SPLINE
SPL {X  -126.418, Y  +769.557, Z    +0.000, E1  +417.118, E3 -55794.219}
SPL {X  -145.244, Y  +738.589, Z    +0.000, E1  +410.405, E3 -55807.461}
SPL {X  -150.151, Y  +726.741, Z    +0.000, E1  +406.068, E3 -55810.388}
SPL {X  -156.642, Y  +704.059, Z    +0.000, E1  +393.659, E3 -55814.017}
SPL {X  -159.317, Y  +686.157, Z    +0.000, E1  +378.660, E3 -55815.507}
SPL {X  -159.973, Y  +673.799, Z    +0.000, E1  +365.345, E3 -55815.956}
SPL {X  -159.990, Y  +669.500, Z    +0.000, E1  +360.000, E3 -55815.996}
SPL {X  -159.990, Y  +667.794, Z    +0.000, E1  +355.745, E3 -55816.007}
SPL {X  -159.990, Y  +664.091, Z    +0.000, E1  +345.072, E3 -55816.079}
SPL {X  -159.990, Y  +659.599, Z    +0.000, E1  +331.984, E3 -55816.250}
SPL {X  -159.990, Y  +652.711, Z    +0.000, E1  +315.707, E3 -55816.729}
SPL {X  -159.990, Y  +640.730, Z    +0.000, E1  +299.703, E3 -55818.078}
SPL {X  -159.990, Y  +620.478, Z    +0.000, E1  +289.974, E3 -55821.891}
SPL {X  -159.990, Y  +573.021, Z    +0.000, E1  +285.381, E3 -55835.835}
SPL {X  -155.476, Y  +344.766, Z    +0.000, E1  +283.975, E3 -55927.806}
SPL {X  -153.405, Y  +337.073, Z    +0.000, E1  +284.153, E3 -55933.861}
SPL {X  -150.223, Y  +327.456, Z    +0.000, E1  +284.427, E3 -55941.947}
SPL {X  -136.549, Y  +299.126, Z    +0.000, E1  +282.463, E3 -55934.837}
ENDSPLINE

SPLINE
SPL {X  -136.626, Y  +299.252, Z    +0.000, E1  +283.686, E3 -55946.487}
ENDSPLINE

SPLINE
SPL {X  -135.890, Y  +298.057, Z    +0.000, E1  +284.960, E3 -55957.836}
SPL {X  -134.349, Y  +295.626, Z    +0.000, E1  +285.678, E3 -55964.683}
SPL {X  -131.287, Y  +291.064, Z    +0.000, E1  +286.028, E3 -55969.496}
SPL {X  -128.265, Y  +286.871, Z    +0.000, E1  +286.387, E3 -55973.952}
SPL {X  -125.161, Y  +282.843, Z    +0.000, E1  +286.768, E3 -55978.224}
SPL {X  -122.038, Y  +279.042, Z    +0.000, E1  +287.168, E3 -55982.204}
SPL {X  -118.642, Y  +275.165, Z    +0.000, E1  +287.619, E3 -55986.167}
SPL {X   -66.040, Y  +236.776, Z    +0.000, E1  +304.306, E3 -56147.530}
ENDSPLINE

SPLINE
SPL {X  -127.452, Y  +285.790, Z    +0.000, E1  +303.409, E3 -56321.476}
SPL {X  -148.001, Y  +321.733, Z    +0.000, E1  +312.190, E3 -56335.579}
SPL {X  -154.604, Y  +341.337, Z    +0.000, E1  +321.370, E3 -56339.353}
SPL {X  -158.135, Y  +358.205, Z    +0.000, E1  +333.016, E3 -56341.302}
SPL {X  -159.602, Y  +371.361, Z    +0.000, E1  +345.165, E3 -56342.198}
SPL {X  -159.981, Y  +380.818, Z    +0.000, E1  +355.488, E3 -56342.476}
SPL {X  -159.990, Y  +384.681, Z    +0.000, E1  +360.222, E3 -56342.505}
SPL {X  -159.990, Y  +389.079, Z    +0.000, E1  +372.017, E3 -56342.568}
SPL {X  -159.990, Y  +394.216, Z    +0.000, E1  +387.062, E3 -56342.760}
SPL {X  -159.990, Y  +401.720, Z    +0.000, E1  +404.434, E3 -56343.303}
SPL {X  -159.990, Y  +414.231, Z    +0.000, E1  +420.575, E3 -56344.832}
SPL {X  -159.990, Y  +462.953, Z    +0.000, E1  +433.611, E3 -56356.571}
SPL {X  -153.839, Y  +715.436, Z    +0.000, E1  +435.884, E3 -56459.002}
SPL {X  -149.923, Y  +727.355, Z    +0.000, E1  +435.515, E3 -56469.112}
SPL {X  -145.995, Y  +736.939, Z    +0.000, E1  +435.150, E3 -56477.846}
SPL {X  -142.305, Y  +744.618, Z    +0.000, E1  +434.773, E3 -56485.290}
SPL {X  -139.557, Y  +749.735, Z    +0.000, E1  +434.483, E3 -56490.439}
SPL {X  -136.371, Y  +755.165, Z    +0.000, E1  +434.152, E3 -56495.984}
SPL {X  -133.102, Y  +760.274, Z    +0.000, E1  +433.777, E3 -56501.369}
SPL {X  -128.975, Y  +766.169, Z    +0.000, E1  +433.313, E3 -56507.645}
SPL {X  -124.947, Y  +771.425, Z    +0.000, E1  +432.782, E3 -56513.338}
SPL {X  -121.698, Y  +775.357, Z    +0.000, E1  +432.353, E3 -56517.532}
SPL {X  -118.622, Y  +778.858, Z    +0.000, E1  +431.924, E3 -56521.158}
SPL {X   -66.171, Y  +817.165, Z    +0.000, E1  +416.016, E3 -56672.517}
ENDSPLINE

SPLINE
SPL {X  -126.418, Y  +769.557, Z    +0.000, E1  +417.118, E3 -56855.758}
SPL {X  -145.244, Y  +738.589, Z    +0.000, E1  +410.405, E3 -56868.999}
SPL {X  -150.151, Y  +726.741, Z    +0.000, E1  +406.068, E3 -56871.926}
SPL {X  -156.642, Y  +704.059, Z    +0.000, E1  +393.659, E3 -56875.555}
SPL {X  -159.317, Y  +686.157, Z    +0.000, E1  +378.660, E3 -56877.046}
SPL {X  -159.973, Y  +673.799, Z    +0.000, E1  +365.345, E3 -56877.494}
SPL {X  -159.990, Y  +669.500, Z    +0.000, E1  +360.000, E3 -56877.534}
SPL {X  -159.990, Y  +667.794, Z    +0.000, E1  +355.745, E3 -56877.546}
SPL {X  -159.990, Y  +664.091, Z    +0.000, E1  +345.072, E3 -56877.618}
SPL {X  -159.990, Y  +658.301, Z    +0.000, E1  +328.717, E3 -56877.870}
SPL {X  -159.990, Y  +650.845, Z    +0.000, E1  +312.108, E3 -56878.415}
SPL {X  -159.990, Y  +640.730, Z    +0.000, E1  +299.703, E3 -56879.617}
SPL {X  -159.990, Y  +620.478, Z    +0.000, E1  +289.974, E3 -56883.430}
SPL {X  -159.990, Y  +573.021, Z    +0.000, E1  +285.381, E3 -56897.374}
SPL {X  -154.165, Y  +339.724, Z    +0.000, E1  +284.073, E3 -56993.221}
SPL {X  -150.223, Y  +327.456, Z    +0.000, E1  +284.427, E3 -57003.486}
SPL {X  -136.549, Y  +299.126, Z    +0.000, E1  +282.463, E3 -56996.376}
ENDSPLINE

SPLINE
SPL {X  -136.862, Y  +299.641, Z    +0.000, E1  +283.396, E3 -57005.018}
ENDSPLINE

SPLINE
SPL {X  -136.434, Y  +298.938, Z    +0.000, E1  +284.018, E3 -57010.909}
SPL {X  -135.890, Y  +298.057, Z    +0.000, E1  +284.960, E3 -57019.375}
SPL {X  -134.349, Y  +295.626, Z    +0.000, E1  +285.678, E3 -57026.222}
SPL {X  -131.287, Y  +291.064, Z    +0.000, E1  +286.028, E3 -57031.034}
SPL {X  -128.265, Y  +286.871, Z    +0.000, E1  +286.387, E3 -57035.490}
SPL {X  -125.161, Y  +282.843, Z    +0.000, E1  +286.768, E3 -57039.762}
SPL {X  -122.038, Y  +279.042, Z    +0.000, E1  +287.168, E3 -57043.742}
SPL {X  -118.642, Y  +275.165, Z    +0.000, E1  +287.619, E3 -57047.705}
SPL {X   -66.040, Y  +236.776, Z    +0.000, E1  +304.306, E3 -57209.069}
ENDSPLINE

SPLINE
SPL {X  -127.452, Y  +285.790, Z    +0.000, E1  +303.409, E3 -57383.014}
SPL {X  -148.001, Y  +321.733, Z    +0.000, E1  +312.190, E3 -57397.118}
SPL {X  -154.604, Y  +341.337, Z    +0.000, E1  +321.370, E3 -57400.891}
SPL {X  -158.135, Y  +358.205, Z    +0.000, E1  +333.016, E3 -57402.841}
SPL {X  -159.602, Y  +371.361, Z    +0.000, E1  +345.165, E3 -57403.737}
SPL {X  -159.981, Y  +380.818, Z    +0.000, E1  +355.488, E3 -57404.015}
SPL {X  -159.990, Y  +384.681, Z    +0.000, E1  +360.222, E3 -57404.044}
SPL {X  -159.990, Y  +389.079, Z    +0.000, E1  +372.017, E3 -57404.107}
SPL {X  -159.990, Y  +394.216, Z    +0.000, E1  +387.062, E3 -57404.299}
SPL {X  -159.990, Y  +399.855, Z    +0.000, E1  +400.916, E3 -57404.670}
SPL {X  -159.990, Y  +405.475, Z    +0.000, E1  +411.039, E3 -57405.187}
SPL {X  -159.990, Y  +414.231, Z    +0.000, E1  +420.575, E3 -57406.371}
SPL {X  -159.990, Y  +462.953, Z    +0.000, E1  +433.611, E3 -57418.110}
SPL {X  -153.839, Y  +715.436, Z    +0.000, E1  +435.884, E3 -57520.540}
SPL {X  -148.840, Y  +730.182, Z    +0.000, E1  +435.434, E3 -57533.117}
SPL {X  -143.409, Y  +742.426, Z    +0.000, E1  +434.905, E3 -57544.629}
SPL {X  -139.557, Y  +749.735, Z    +0.000, E1  +434.483, E3 -57551.977}
SPL {X  -136.371, Y  +755.165, Z    +0.000, E1  +434.152, E3 -57557.523}
SPL {X  -133.102, Y  +760.274, Z    +0.000, E1  +433.777, E3 -57562.908}
SPL {X  -128.975, Y  +766.169, Z    +0.000, E1  +433.313, E3 -57569.183}
SPL {X  -124.947, Y  +771.425, Z    +0.000, E1  +432.782, E3 -57574.876}
SPL {X  -121.698, Y  +775.357, Z    +0.000, E1  +432.353, E3 -57579.071}
SPL {X  -118.622, Y  +778.858, Z    +0.000, E1  +431.924, E3 -57582.697}
SPL {X   -66.171, Y  +817.165, Z    +0.000, E1  +416.016, E3 -57734.055}
ENDSPLINE

SPLINE
SPL {X  -126.418, Y  +769.557, Z    +0.000, E1  +417.118, E3 -57917.296}
SPL {X  -145.244, Y  +738.589, Z    +0.000, E1  +410.405, E3 -57930.538}
SPL {X  -150.151, Y  +726.741, Z    +0.000, E1  +406.068, E3 -57933.464}
SPL {X  -156.642, Y  +704.059, Z    +0.000, E1  +393.659, E3 -57937.094}
SPL {X  -159.317, Y  +686.157, Z    +0.000, E1  +378.660, E3 -57938.584}
SPL {X  -159.973, Y  +673.799, Z    +0.000, E1  +365.345, E3 -57939.033}
SPL {X  -159.990, Y  +669.500, Z    +0.000, E1  +360.000, E3 -57939.073}
SPL {X  -159.990, Y  +667.794, Z    +0.000, E1  +355.745, E3 -57939.084}
SPL {X  -159.990, Y  +664.091, Z    +0.000, E1  +345.072, E3 -57939.156}
SPL {X  -159.990, Y  +658.301, Z    +0.000, E1  +328.717, E3 -57939.409}
SPL {X  -159.990, Y  +650.845, Z    +0.000, E1  +312.108, E3 -57939.954}
SPL {X  -159.990, Y  +640.730, Z    +0.000, E1  +299.703, E3 -57941.155}
SPL {X  -159.990, Y  +620.478, Z    +0.000, E1  +289.974, E3 -57944.968}
SPL {X  -159.990, Y  +573.021, Z    +0.000, E1  +285.381, E3 -57958.912}
SPL {X  -154.165, Y  +339.724, Z    +0.000, E1  +284.073, E3 -58054.759}
SPL {X  -150.223, Y  +327.456, Z    +0.000, E1  +284.427, E3 -58065.024}
SPL {X  -136.549, Y  +299.126, Z    +0.000, E1  +282.463, E3 -58057.914}
ENDSPLINE

SPLINE
SPL {X  -136.862, Y  +299.641, Z    +0.000, E1  +283.396, E3 -58066.556}
ENDSPLINE

SPLINE
SPL {X  -136.434, Y  +298.938, Z    +0.000, E1  +284.018, E3 -58072.447}
SPL {X  -135.890, Y  +298.057, Z    +0.000, E1  +284.960, E3 -58080.913}
SPL {X  -134.349, Y  +295.626, Z    +0.000, E1  +285.678, E3 -58087.760}
SPL {X  -131.287, Y  +291.064, Z    +0.000, E1  +286.028, E3 -58092.573}
SPL {X  -128.265, Y  +286.871, Z    +0.000, E1  +286.387, E3 -58097.029}
SPL {X  -125.161, Y  +282.843, Z    +0.000, E1  +286.768, E3 -58101.301}
SPL {X  -122.038, Y  +279.042, Z    +0.000, E1  +287.168, E3 -58105.281}
SPL {X  -118.642, Y  +275.165, Z    +0.000, E1  +287.619, E3 -58109.244}
SPL {X   -66.040, Y  +236.776, Z    +0.000, E1  +304.306, E3 -58270.607}
ENDSPLINE

SPLINE
SPL {X  -127.452, Y  +285.790, Z    +0.000, E1  +303.409, E3 -58444.552}
SPL {X  -148.001, Y  +321.733, Z    +0.000, E1  +312.190, E3 -58458.656}
SPL {X  -154.604, Y  +341.337, Z    +0.000, E1  +321.370, E3 -58462.430}
SPL {X  -158.135, Y  +358.205, Z    +0.000, E1  +333.016, E3 -58464.379}
SPL {X  -159.602, Y  +371.361, Z    +0.000, E1  +345.165, E3 -58465.275}
SPL {X  -159.981, Y  +380.818, Z    +0.000, E1  +355.488, E3 -58465.553}
SPL {X  -159.990, Y  +384.681, Z    +0.000, E1  +360.222, E3 -58465.582}
SPL {X  -159.990, Y  +389.079, Z    +0.000, E1  +372.017, E3 -58465.645}
SPL {X  -159.990, Y  +394.216, Z    +0.000, E1  +387.062, E3 -58465.837}
SPL {X  -159.990, Y  +399.855, Z    +0.000, E1  +400.916, E3 -58466.208}
SPL {X  -159.990, Y  +405.475, Z    +0.000, E1  +411.039, E3 -58466.725}
SPL {X  -159.990, Y  +414.231, Z    +0.000, E1  +420.575, E3 -58467.909}
SPL {X  -159.990, Y  +462.953, Z    +0.000, E1  +433.611, E3 -58479.648}
SPL {X  -153.839, Y  +715.436, Z    +0.000, E1  +435.884, E3 -58582.079}
SPL {X  -148.840, Y  +730.182, Z    +0.000, E1  +435.434, E3 -58594.655}
SPL {X  -143.409, Y  +742.426, Z    +0.000, E1  +434.905, E3 -58606.167}
SPL {X  -139.557, Y  +749.735, Z    +0.000, E1  +434.483, E3 -58613.515}
SPL {X  -136.371, Y  +755.165, Z    +0.000, E1  +434.152, E3 -58619.061}
SPL {X  -133.102, Y  +760.274, Z    +0.000, E1  +433.777, E3 -58624.446}
SPL {X  -128.975, Y  +766.169, Z    +0.000, E1  +433.313, E3 -58630.722}
SPL {X  -124.947, Y  +771.425, Z    +0.000, E1  +432.782, E3 -58636.415}
SPL {X  -121.698, Y  +775.357, Z    +0.000, E1  +432.353, E3 -58640.609}
SPL {X  -118.622, Y  +778.858, Z    +0.000, E1  +431.924, E3 -58644.235}
SPL {X   -66.171, Y  +817.165, Z    +0.000, E1  +416.016, E3 -58795.593}
ENDSPLINE

SPLINE
SPL {X  -126.418, Y  +769.557, Z    +0.000, E1  +417.118, E3 -58978.835}
SPL {X  -145.244, Y  +738.589, Z    +0.000, E1  +410.405, E3 -58992.076}
SPL {X  -150.151, Y  +726.741, Z    +0.000, E1  +406.068, E3 -58995.003}
SPL {X  -156.642, Y  +704.059, Z    +0.000, E1  +393.659, E3 -58998.632}
SPL {X  -159.317, Y  +686.157, Z    +0.000, E1  +378.660, E3 -59000.123}
SPL {X  -159.973, Y  +673.799, Z    +0.000, E1  +365.345, E3 -59000.571}
SPL {X  -159.990, Y  +669.500, Z    +0.000, E1  +360.000, E3 -59000.611}
SPL {X  -159.990, Y  +667.794, Z    +0.000, E1  +355.745, E3 -59000.623}
SPL {X  -159.990, Y  +664.091, Z    +0.000, E1  +345.072, E3 -59000.695}
SPL {X  -159.990, Y  +658.301, Z    +0.000, E1  +328.717, E3 -59000.947}
SPL {X  -159.990, Y  +650.845, Z    +0.000, E1  +312.108, E3 -59001.492}
SPL {X  -159.990, Y  +640.730, Z    +0.000, E1  +299.703, E3 -59002.693}
SPL {X  -159.990, Y  +620.478, Z    +0.000, E1  +289.974, E3 -59006.507}
SPL {X  -159.990, Y  +573.021, Z    +0.000, E1  +285.381, E3 -59020.451}
SPL {X  -154.165, Y  +339.724, Z    +0.000, E1  +284.073, E3 -59116.298}
SPL {X  -150.223, Y  +327.456, Z    +0.000, E1  +284.427, E3 -59126.562}
SPL {X  -136.549, Y  +299.126, Z    +0.000, E1  +282.463, E3 -59119.452}
ENDSPLINE

SPLINE
SPL {X  -136.862, Y  +299.641, Z    +0.000, E1  +283.396, E3 -59128.094}
ENDSPLINE

SPLINE
SPL {X  -136.434, Y  +298.938, Z    +0.000, E1  +284.018, E3 -59133.986}
SPL {X  -135.890, Y  +298.057, Z    +0.000, E1  +284.960, E3 -59142.452}
SPL {X  -134.349, Y  +295.626, Z    +0.000, E1  +285.678, E3 -59149.299}
SPL {X  -131.287, Y  +291.064, Z    +0.000, E1  +286.028, E3 -59154.111}
SPL {X  -128.265, Y  +286.871, Z    +0.000, E1  +286.387, E3 -59158.567}
SPL {X  -125.161, Y  +282.843, Z    +0.000, E1  +286.768, E3 -59162.839}
SPL {X  -122.038, Y  +279.042, Z    +0.000, E1  +287.168, E3 -59166.819}
SPL {X  -118.642, Y  +275.165, Z    +0.000, E1  +287.619, E3 -59170.782}
SPL {X   -66.040, Y  +236.776, Z    +0.000, E1  +304.306, E3 -59332.146}
ENDSPLINE

SPLINE
SPL {X  -127.452, Y  +285.790, Z    +0.000, E1  +303.409, E3 -59506.091}
SPL {X  -151.591, Y  +331.344, Z    +0.000, E1  +316.130, E3 -59522.190}
SPL {X  -158.135, Y  +358.205, Z    +0.000, E1  +333.016, E3 -59525.918}
SPL {X  -159.602, Y  +371.361, Z    +0.000, E1  +345.165, E3 -59526.814}
SPL {X  -159.981, Y  +380.818, Z    +0.000, E1  +355.488, E3 -59527.092}
SPL {X  -159.990, Y  +384.681, Z    +0.000, E1  +360.222, E3 -59527.121}
SPL {X  -159.990, Y  +387.626, Z    +0.000, E1  +368.190, E3 -59527.149}
SPL {X  -159.990, Y  +390.340, Z    +0.000, E1  +375.987, E3 -59527.214}
SPL {X  -159.990, Y  +394.216, Z    +0.000, E1  +387.062, E3 -59527.375}
SPL {X  -159.990, Y  +399.855, Z    +0.000, E1  +400.916, E3 -59527.747}
SPL {X  -159.990, Y  +405.475, Z    +0.000, E1  +411.039, E3 -59528.263}
SPL {X  -159.990, Y  +414.231, Z    +0.000, E1  +420.575, E3 -59529.448}
SPL {X  -159.990, Y  +462.953, Z    +0.000, E1  +433.611, E3 -59541.187}
SPL {X  -153.839, Y  +715.436, Z    +0.000, E1  +435.884, E3 -59643.617}
SPL {X  -148.840, Y  +730.182, Z    +0.000, E1  +435.434, E3 -59656.194}
SPL {X  -143.409, Y  +742.426, Z    +0.000, E1  +434.905, E3 -59667.706}
SPL {X  -139.557, Y  +749.735, Z    +0.000, E1  +434.483, E3 -59675.054}
SPL {X  -136.371, Y  +755.165, Z    +0.000, E1  +434.152, E3 -59680.600}
SPL {X  -133.102, Y  +760.274, Z    +0.000, E1  +433.777, E3 -59685.985}
SPL {X  -128.975, Y  +766.169, Z    +0.000, E1  +433.313, E3 -59692.260}
SPL {X  -124.947, Y  +771.425, Z    +0.000, E1  +432.782, E3 -59697.953}
SPL {X  -121.698, Y  +775.357, Z    +0.000, E1  +432.353, E3 -59702.148}
SPL {X  -118.622, Y  +778.858, Z    +0.000, E1  +431.924, E3 -59705.774}
SPL {X   -66.171, Y  +817.165, Z    +0.000, E1  +416.016, E3 -59857.132}
ENDSPLINE

SPLINE
SPL {X  -126.418, Y  +769.557, Z    +0.000, E1  +417.118, E3 -60040.373}
SPL {X  -148.476, Y  +731.097, Z    +0.000, E1  +407.824, E3 -60055.529}
SPL {X  -156.642, Y  +704.059, Z    +0.000, E1  +393.659, E3 -60060.171}
SPL {X  -159.317, Y  +686.157, Z    +0.000, E1  +378.660, E3 -60061.661}
SPL {X  -159.907, Y  +676.666, Z    +0.000, E1  +368.555, E3 -60062.059}
SPL {X  -159.990, Y  +669.586, Z    +0.000, E1  +360.216, E3 -60062.149}
SPL {X  -159.990, Y  +667.794, Z    +0.000, E1  +355.745, E3 -60062.161}
SPL {X  -159.990, Y  +664.091, Z    +0.000, E1  +345.072, E3 -60062.233}
SPL {X  -159.990, Y  +659.599, Z    +0.000, E1  +331.984, E3 -60062.404}
SPL {X  -159.990, Y  +652.711, Z    +0.000, E1  +315.707, E3 -60062.883}
SPL {X  -159.990, Y  +640.730, Z    +0.000, E1  +299.703, E3 -60064.232}
SPL {X  -159.990, Y  +620.478, Z    +0.000, E1  +289.974, E3 -60068.045}
SPL {X  -159.990, Y  +573.021, Z    +0.000, E1  +285.381, E3 -60081.989}
SPL {X  -154.165, Y  +339.724, Z    +0.000, E1  +284.073, E3 -60177.836}
SPL {X  -150.571, Y  +328.416, Z    +0.000, E1  +284.401, E3 -60187.281}
SPL {X  -148.206, Y  +322.236, Z    +0.000, E1  +284.635, E3 -60192.826}
SPL {X  -136.549, Y  +299.126, Z    +0.000, E1  +282.463, E3 -60180.991}
ENDSPLINE

SPLINE
SPL {X  -136.862, Y  +299.641, Z    +0.000, E1  +283.396, E3 -60189.633}
ENDSPLINE

SPLINE
SPL {X  -136.434, Y  +298.938, Z    +0.000, E1  +284.018, E3 -60195.524}
SPL {X  -135.890, Y  +298.057, Z    +0.000, E1  +284.960, E3 -60203.990}
SPL {X  -134.349, Y  +295.626, Z    +0.000, E1  +285.678, E3 -60210.837}
SPL {X  -131.287, Y  +291.064, Z    +0.000, E1  +286.028, E3 -60215.650}
SPL {X  -128.265, Y  +286.871, Z    +0.000, E1  +286.387, E3 -60220.106}
SPL {X  -125.161, Y  +282.843, Z    +0.000, E1  +286.768, E3 -60224.378}
SPL {X  -122.038, Y  +279.042, Z    +0.000, E1  +287.168, E3 -60228.357}
SPL {X  -118.642, Y  +275.165, Z    +0.000, E1  +287.619, E3 -60232.321}
SPL {X   -66.040, Y  +236.776, Z    +0.000, E1  +304.306, E3 -60393.684}
ENDSPLINE

SPLINE
SPL {X  -127.452, Y  +285.790, Z    +0.000, E1  +303.409, E3 -60567.629}
SPL {X  -151.591, Y  +331.344, Z    +0.000, E1  +316.130, E3 -60583.729}
SPL {X  -158.135, Y  +358.205, Z    +0.000, E1  +333.016, E3 -60587.456}
SPL {X  -159.602, Y  +371.361, Z    +0.000, E1  +345.165, E3 -60588.352}
SPL {X  -159.981, Y  +380.818, Z    +0.000, E1  +355.488, E3 -60588.630}
SPL {X  -159.990, Y  +384.681, Z    +0.000, E1  +360.222, E3 -60588.659}
SPL {X  -159.990, Y  +389.079, Z    +0.000, E1  +372.017, E3 -60588.722}
SPL {X  -159.990, Y  +394.216, Z    +0.000, E1  +387.062, E3 -60588.914}
SPL {X  -159.990, Y  +399.855, Z    +0.000, E1  +400.916, E3 -60589.285}
SPL {X  -159.990, Y  +405.475, Z    +0.000, E1  +411.039, E3 -60589.802}
SPL {X  -159.990, Y  +414.231, Z    +0.000, E1  +420.575, E3 -60590.986}
SPL {X  -159.990, Y  +462.953, Z    +0.000, E1  +433.611, E3 -60602.725}
SPL {X  -153.839, Y  +715.436, Z    +0.000, E1  +435.884, E3 -60705.156}
SPL {X  -148.840, Y  +730.182, Z    +0.000, E1  +435.434, E3 -60717.732}
SPL {X  -143.409, Y  +742.426, Z    +0.000, E1  +434.905, E3 -60729.244}
SPL {X  -139.557, Y  +749.735, Z    +0.000, E1  +434.483, E3 -60736.592}
SPL {X  -136.371, Y  +755.165, Z    +0.000, E1  +434.152, E3 -60742.138}
SPL {X  -133.102, Y  +760.274, Z    +0.000, E1  +433.777, E3 -60747.523}
SPL {X  -128.975, Y  +766.169, Z    +0.000, E1  +433.313, E3 -60753.799}
SPL {X  -124.947, Y  +771.425, Z    +0.000, E1  +432.782, E3 -60759.492}
SPL {X  -121.698, Y  +775.357, Z    +0.000, E1  +432.353, E3 -60763.686}
SPL {X  -118.622, Y  +778.858, Z    +0.000, E1  +431.924, E3 -60767.312}
SPL {X   -66.171, Y  +817.165, Z    +0.000, E1  +416.016, E3 -60918.670}
ENDSPLINE

SPLINE
SPL {X  -126.418, Y  +769.557, Z    +0.000, E1  +417.118, E3 -61101.912}
SPL {X  -145.244, Y  +738.589, Z    +0.000, E1  +410.405, E3 -61115.153}
SPL {X  -150.151, Y  +726.741, Z    +0.000, E1  +406.068, E3 -61118.080}
SPL {X  -156.642, Y  +704.059, Z    +0.000, E1  +393.659, E3 -61121.709}
SPL {X  -159.317, Y  +686.157, Z    +0.000, E1  +378.660, E3 -61123.200}
SPL {X  -159.973, Y  +673.799, Z    +0.000, E1  +365.345, E3 -61123.648}
SPL {X  -159.990, Y  +669.500, Z    +0.000, E1  +360.000, E3 -61123.688}
SPL {X  -159.990, Y  +667.794, Z    +0.000, E1  +355.745, E3 -61123.699}
SPL {X  -159.990, Y  +664.091, Z    +0.000, E1  +345.072, E3 -61123.772}
SPL {X  -159.990, Y  +658.301, Z    +0.000, E1  +328.717, E3 -61124.024}
SPL {X  -159.990, Y  +650.845, Z    +0.000, E1  +312.108, E3 -61124.569}
SPL {X  -159.990, Y  +640.730, Z    +0.000, E1  +299.703, E3 -61125.770}
SPL {X  -159.990, Y  +620.478, Z    +0.000, E1  +289.974, E3 -61129.584}
SPL {X  -159.990, Y  +573.021, Z    +0.000, E1  +285.381, E3 -61143.528}
SPL {X  -154.165, Y  +339.724, Z    +0.000, E1  +284.073, E3 -61239.374}
SPL {X  -150.223, Y  +327.456, Z    +0.000, E1  +284.427, E3 -61249.639}
SPL {X  -136.549, Y  +299.126, Z    +0.000, E1  +282.463, E3 -61242.529}
ENDSPLINE

SPLINE
SPL {X  -136.862, Y  +299.641, Z    +0.000, E1  +283.396, E3 -61251.171}
ENDSPLINE

SPLINE
SPL {X  -136.434, Y  +298.938, Z    +0.000, E1  +284.018, E3 -61257.062}
SPL {X  -135.890, Y  +298.057, Z    +0.000, E1  +284.960, E3 -61265.528}
SPL {X  -134.349, Y  +295.626, Z    +0.000, E1  +285.678, E3 -61272.376}
SPL {X  -131.287, Y  +291.064, Z    +0.000, E1  +286.028, E3 -61277.188}
SPL {X  -128.265, Y  +286.871, Z    +0.000, E1  +286.387, E3 -61281.644}
SPL {X  -125.161, Y  +282.843, Z    +0.000, E1  +286.768, E3 -61285.916}
SPL {X  -122.038, Y  +279.042, Z    +0.000, E1  +287.168, E3 -61289.896}
SPL {X  -118.642, Y  +275.165, Z    +0.000, E1  +287.619, E3 -61293.859}
SPL {X   -66.040, Y  +236.776, Z    +0.000, E1  +304.306, E3 -61455.223}
ENDSPLINE

SPLINE
SPL {X  -127.452, Y  +285.790, Z    +0.000, E1  +303.409, E3 -61629.168}
SPL {X  -151.591, Y  +331.344, Z    +0.000, E1  +316.130, E3 -61645.267}
SPL {X  -158.135, Y  +358.205, Z    +0.000, E1  +333.016, E3 -61648.995}
SPL {X  -159.602, Y  +371.361, Z    +0.000, E1  +345.165, E3 -61649.891}
SPL {X  -159.981, Y  +380.818, Z    +0.000, E1  +355.488, E3 -61650.169}
SPL {X  -159.990, Y  +384.681, Z    +0.000, E1  +360.222, E3 -61650.198}
SPL {X  -159.990, Y  +387.626, Z    +0.000, E1  +368.190, E3 -61650.226}
SPL {X  -159.990, Y  +390.340, Z    +0.000, E1  +375.987, E3 -61650.290}
SPL {X  -159.990, Y  +394.216, Z    +0.000, E1  +387.062, E3 -61650.452}
SPL {X  -159.990, Y  +399.855, Z    +0.000, E1  +400.916, E3 -61650.823}
SPL {X  -159.990, Y  +405.475, Z    +0.000, E1  +411.039, E3 -61651.340}
SPL {X  -159.990, Y  +414.231, Z    +0.000, E1  +420.575, E3 -61652.525}
SPL {X  -159.990, Y  +462.953, Z    +0.000, E1  +433.611, E3 -61664.264}
SPL {X  -153.839, Y  +715.436, Z    +0.000, E1  +435.884, E3 -61766.694}
SPL {X  -148.840, Y  +730.182, Z    +0.000, E1  +435.434, E3 -61779.271}
SPL {X  -143.409, Y  +742.426, Z    +0.000, E1  +434.905, E3 -61790.783}
SPL {X  -139.557, Y  +749.735, Z    +0.000, E1  +434.483, E3 -61798.131}
SPL {X  -136.371, Y  +755.165, Z    +0.000, E1  +434.152, E3 -61803.677}
SPL {X  -133.102, Y  +760.274, Z    +0.000, E1  +433.777, E3 -61809.062}
SPL {X  -128.975, Y  +766.169, Z    +0.000, E1  +433.313, E3 -61815.337}
SPL {X  -124.947, Y  +771.425, Z    +0.000, E1  +432.782, E3 -61821.030}
SPL {X  -121.698, Y  +775.357, Z    +0.000, E1  +432.353, E3 -61825.225}
SPL {X  -118.622, Y  +778.858, Z    +0.000, E1  +431.924, E3 -61828.851}
SPL {X   -66.171, Y  +817.165, Z    +0.000, E1  +416.016, E3 -61980.209}
ENDSPLINE

SPLINE
SPL {X  -126.418, Y  +769.557, Z    +0.000, E1  +417.118, E3 -62163.450}
SPL {X  -148.476, Y  +731.097, Z    +0.000, E1  +407.824, E3 -62178.606}
SPL {X  -156.642, Y  +704.059, Z    +0.000, E1  +393.659, E3 -62183.248}
SPL {X  -159.317, Y  +686.157, Z    +0.000, E1  +378.660, E3 -62184.738}
SPL {X  -159.973, Y  +673.799, Z    +0.000, E1  +365.345, E3 -62185.187}
SPL {X  -159.990, Y  +669.500, Z    +0.000, E1  +360.000, E3 -62185.227}
SPL {X  -159.990, Y  +667.794, Z    +0.000, E1  +355.745, E3 -62185.238}
SPL {X  -159.990, Y  +664.091, Z    +0.000, E1  +345.072, E3 -62185.310}
SPL {X  -159.990, Y  +659.599, Z    +0.000, E1  +331.984, E3 -62185.480}
SPL {X  -159.990, Y  +652.711, Z    +0.000, E1  +315.707, E3 -62185.960}
SPL {X  -159.990, Y  +640.730, Z    +0.000, E1  +299.703, E3 -62187.309}
SPL {X  -159.990, Y  +620.478, Z    +0.000, E1  +289.974, E3 -62191.122}
SPL {X  -159.990, Y  +573.021, Z    +0.000, E1  +285.381, E3 -62205.066}
SPL {X  -154.165, Y  +339.724, Z    +0.000, E1  +284.073, E3 -62300.913}
SPL {X  -150.223, Y  +327.456, Z    +0.000, E1  +284.427, E3 -62311.178}
SPL {X  -136.549, Y  +299.126, Z    +0.000, E1  +282.463, E3 -62304.068}
ENDSPLINE

SPLINE
SPL {X  -136.862, Y  +299.641, Z    +0.000, E1  +283.396, E3 -62312.710}
ENDSPLINE

SPLINE
SPL {X  -136.434, Y  +298.938, Z    +0.000, E1  +284.018, E3 -62318.601}
SPL {X  -135.890, Y  +298.057, Z    +0.000, E1  +284.960, E3 -62327.067}
SPL {X  -134.349, Y  +295.626, Z    +0.000, E1  +285.678, E3 -62333.914}
SPL {X  -131.287, Y  +291.064, Z    +0.000, E1  +286.028, E3 -62338.727}
SPL {X  -128.265, Y  +286.871, Z    +0.000, E1  +286.387, E3 -62343.183}
SPL {X  -125.161, Y  +282.843, Z    +0.000, E1  +286.768, E3 -62347.454}
SPL {X  -122.038, Y  +279.042, Z    +0.000, E1  +287.168, E3 -62351.434}
SPL {X  -118.642, Y  +275.165, Z    +0.000, E1  +287.619, E3 -62355.398}
SPL {X   -66.040, Y  +236.776, Z    +0.000, E1  +304.306, E3 -62516.761}
ENDSPLINE

SPLINE
SPL {X  -127.452, Y  +285.790, Z    +0.000, E1  +303.409, E3 -62690.706}
SPL {X  -151.591, Y  +331.344, Z    +0.000, E1  +316.130, E3 -62706.806}
SPL {X  -158.135, Y  +358.205, Z    +0.000, E1  +333.016, E3 -62710.533}
SPL {X  -159.602, Y  +371.361, Z    +0.000, E1  +345.165, E3 -62711.429}
SPL {X  -159.981, Y  +380.818, Z    +0.000, E1  +355.488, E3 -62711.707}
SPL {X  -159.990, Y  +384.681, Z    +0.000, E1  +360.222, E3 -62711.736}
SPL {X  -159.990, Y  +387.626, Z    +0.000, E1  +368.190, E3 -62711.764}
SPL {X  -159.990, Y  +390.340, Z    +0.000, E1  +375.987, E3 -62711.829}
SPL {X  -159.990, Y  +394.216, Z    +0.000, E1  +387.062, E3 -62711.991}
SPL {X  -159.990, Y  +399.855, Z    +0.000, E1  +400.916, E3 -62712.362}
SPL {X  -159.990, Y  +405.475, Z    +0.000, E1  +411.039, E3 -62712.879}
SPL {X  -159.990, Y  +414.231, Z    +0.000, E1  +420.575, E3 -62714.063}
SPL {X  -159.990, Y  +462.953, Z    +0.000, E1  +433.611, E3 -62725.802}
SPL {X  -153.839, Y  +715.436, Z    +0.000, E1  +435.884, E3 -62828.233}
SPL {X  -148.840, Y  +730.182, Z    +0.000, E1  +435.434, E3 -62840.809}
SPL {X  -143.409, Y  +742.426, Z    +0.000, E1  +434.905, E3 -62852.321}
SPL {X  -139.557, Y  +749.735, Z    +0.000, E1  +434.483, E3 -62859.669}
SPL {X  -136.371, Y  +755.165, Z    +0.000, E1  +434.152, E3 -62865.215}
SPL {X  -133.102, Y  +760.274, Z    +0.000, E1  +433.777, E3 -62870.600}
SPL {X  -128.975, Y  +766.169, Z    +0.000, E1  +433.313, E3 -62876.875}
SPL {X  -124.947, Y  +771.425, Z    +0.000, E1  +432.782, E3 -62882.568}
SPL {X  -121.698, Y  +775.357, Z    +0.000, E1  +432.353, E3 -62886.763}
SPL {X  -118.622, Y  +778.858, Z    +0.000, E1  +431.924, E3 -62890.389}
SPL {X   -66.171, Y  +817.165, Z    +0.000, E1  +416.016, E3 -63041.747}
ENDSPLINE

SPLINE
SPL {X  -126.418, Y  +769.557, Z    +0.000, E1  +417.118, E3 -63224.989}
SPL {X  -148.476, Y  +731.097, Z    +0.000, E1  +407.824, E3 -63240.145}
SPL {X  -156.642, Y  +704.059, Z    +0.000, E1  +393.659, E3 -63244.786}
SPL {X  -159.317, Y  +686.157, Z    +0.000, E1  +378.660, E3 -63246.276}
SPL {X  -159.973, Y  +673.799, Z    +0.000, E1  +365.345, E3 -63246.725}
SPL {X  -159.990, Y  +669.500, Z    +0.000, E1  +360.000, E3 -63246.765}
SPL {X  -159.990, Y  +667.794, Z    +0.000, E1  +355.745, E3 -63246.776}
SPL {X  -159.990, Y  +664.091, Z    +0.000, E1  +345.072, E3 -63246.848}
SPL {X  -159.990, Y  +659.599, Z    +0.000, E1  +331.984, E3 -63247.019}
SPL {X  -159.990, Y  +652.711, Z    +0.000, E1  +315.707, E3 -63247.498}
SPL {X  -159.990, Y  +640.730, Z    +0.000, E1  +299.703, E3 -63248.847}
SPL {X  -159.990, Y  +620.478, Z    +0.000, E1  +289.974, E3 -63252.661}
SPL {X  -159.990, Y  +573.021, Z    +0.000, E1  +285.381, E3 -63266.604}
SPL {X  -154.165, Y  +339.724, Z    +0.000, E1  +284.073, E3 -63362.451}
SPL {X  -150.223, Y  +327.456, Z    +0.000, E1  +284.427, E3 -63372.716}
SPL {X  -136.549, Y  +299.126, Z    +0.000, E1  +282.463, E3 -63365.606}
ENDSPLINE

SPLINE
SPL {X  -136.862, Y  +299.641, Z    +0.000, E1  +283.396, E3 -63374.248}
ENDSPLINE

SPLINE
SPL {X  -136.434, Y  +298.938, Z    +0.000, E1  +284.018, E3 -63380.139}
SPL {X  -135.890, Y  +298.057, Z    +0.000, E1  +284.960, E3 -63388.605}
SPL {X  -134.349, Y  +295.626, Z    +0.000, E1  +285.678, E3 -63395.453}
SPL {X  -131.287, Y  +291.064, Z    +0.000, E1  +286.028, E3 -63400.265}
SPL {X  -128.265, Y  +286.871, Z    +0.000, E1  +286.387, E3 -63404.721}
SPL {X  -125.161, Y  +282.843, Z    +0.000, E1  +286.768, E3 -63408.993}
SPL {X  -122.038, Y  +279.042, Z    +0.000, E1  +287.168, E3 -63412.973}
SPL {X  -118.642, Y  +275.165, Z    +0.000, E1  +287.619, E3 -63416.936}
SPL {X   -66.040, Y  +236.776, Z    +0.000, E1  +304.306, E3 -63578.299}
ENDSPLINE

SPLINE
SPL {X  -127.452, Y  +285.790, Z    +0.000, E1  +303.409, E3 -63752.245}
SPL {X  -151.591, Y  +331.344, Z    +0.000, E1  +316.130, E3 -63768.344}
SPL {X  -158.135, Y  +358.205, Z    +0.000, E1  +333.016, E3 -63772.072}
SPL {X  -159.602, Y  +371.361, Z    +0.000, E1  +345.165, E3 -63772.968}
SPL {X  -159.981, Y  +380.818, Z    +0.000, E1  +355.488, E3 -63773.246}
SPL {X  -159.990, Y  +384.681, Z    +0.000, E1  +360.222, E3 -63773.274}
SPL {X  -159.990, Y  +387.626, Z    +0.000, E1  +368.190, E3 -63773.303}
SPL {X  -159.990, Y  +390.340, Z    +0.000, E1  +375.987, E3 -63773.367}
SPL {X  -159.990, Y  +394.216, Z    +0.000, E1  +387.062, E3 -63773.529}
SPL {X  -159.990, Y  +399.855, Z    +0.000, E1  +400.916, E3 -63773.900}
SPL {X  -159.990, Y  +405.475, Z    +0.000, E1  +411.039, E3 -63774.417}
SPL {X  -159.990, Y  +414.231, Z    +0.000, E1  +420.575, E3 -63775.602}
SPL {X  -159.990, Y  +462.953, Z    +0.000, E1  +433.611, E3 -63787.341}
SPL {X  -153.839, Y  +715.436, Z    +0.000, E1  +435.884, E3 -63889.771}
SPL {X  -149.923, Y  +727.355, Z    +0.000, E1  +435.515, E3 -63899.881}
SPL {X  -145.995, Y  +736.939, Z    +0.000, E1  +435.150, E3 -63908.616}
SPL {X  -142.305, Y  +744.618, Z    +0.000, E1  +434.773, E3 -63916.059}
SPL {X  -139.557, Y  +749.735, Z    +0.000, E1  +434.483, E3 -63921.208}
SPL {X  -136.371, Y  +755.165, Z    +0.000, E1  +434.152, E3 -63926.753}
SPL {X  -133.102, Y  +760.274, Z    +0.000, E1  +433.777, E3 -63932.139}
SPL {X  -128.975, Y  +766.169, Z    +0.000, E1  +433.313, E3 -63938.414}
SPL {X  -124.947, Y  +771.425, Z    +0.000, E1  +432.782, E3 -63944.107}
SPL {X  -121.698, Y  +775.357, Z    +0.000, E1  +432.353, E3 -63948.301}
SPL {X  -118.622, Y  +778.858, Z    +0.000, E1  +431.924, E3 -63951.927}
SPL {X   -66.171, Y  +817.165, Z    +0.000, E1  +416.016, E3 -64103.286}
ENDSPLINE

SPLINE
SPL {X  -126.418, Y  +769.557, Z    +0.000, E1  +417.118, E3 -64286.527}
SPL {X  -148.476, Y  +731.097, Z    +0.000, E1  +407.824, E3 -64301.683}
SPL {X  -156.642, Y  +704.059, Z    +0.000, E1  +393.659, E3 -64306.325}
SPL {X  -159.317, Y  +686.157, Z    +0.000, E1  +378.660, E3 -64307.815}
SPL {X  -159.973, Y  +673.799, Z    +0.000, E1  +365.345, E3 -64308.264}
SPL {X  -159.990, Y  +669.500, Z    +0.000, E1  +360.000, E3 -64308.304}
SPL {X  -159.990, Y  +667.794, Z    +0.000, E1  +355.745, E3 -64308.315}
SPL {X  -159.990, Y  +664.091, Z    +0.000, E1  +345.072, E3 -64308.387}
SPL {X  -159.990, Y  +658.301, Z    +0.000, E1  +328.717, E3 -64308.639}
SPL {X  -159.990, Y  +650.845, Z    +0.000, E1  +312.108, E3 -64309.185}
SPL {X  -159.990, Y  +640.730, Z    +0.000, E1  +299.703, E3 -64310.386}
SPL {X  -159.990, Y  +620.478, Z    +0.000, E1  +289.974, E3 -64314.199}
SPL {X  -159.990, Y  +573.021, Z    +0.000, E1  +285.381, E3 -64328.143}
SPL {X  -154.165, Y  +339.724, Z    +0.000, E1  +284.073, E3 -64423.990}
SPL {X  -150.223, Y  +327.456, Z    +0.000, E1  +284.427, E3 -64434.255}
SPL {X  -136.549, Y  +299.126, Z    +0.000, E1  +282.463, E3 -64427.145}
ENDSPLINE

SPLINE
SPL {X  -136.862, Y  +299.641, Z    +0.000, E1  +283.396, E3 -64435.787}
ENDSPLINE

SPLINE
SPL {X  -136.434, Y  +298.938, Z    +0.000, E1  +284.018, E3 -64441.678}
SPL {X  -135.890, Y  +298.057, Z    +0.000, E1  +284.960, E3 -64450.144}
SPL {X  -134.349, Y  +295.626, Z    +0.000, E1  +285.678, E3 -64456.991}
SPL {X  -131.287, Y  +291.064, Z    +0.000, E1  +286.028, E3 -64461.804}
SPL {X  -128.265, Y  +286.871, Z    +0.000, E1  +286.387, E3 -64466.260}
SPL {X  -125.161, Y  +282.843, Z    +0.000, E1  +286.768, E3 -64470.531}
SPL {X  -122.038, Y  +279.042, Z    +0.000, E1  +287.168, E3 -64474.511}
SPL {X  -119.499, Y  +276.120, Z    +0.000, E1  +287.518, E3 -64477.530}
SPL {X  -117.726, Y  +274.160, Z    +0.000, E1  +287.766, E3 -64479.493}
SPL {X   -66.040, Y  +236.776, Z    +0.000, E1  +304.306, E3 -64639.838}
ENDSPLINE

SPLINE
SPL {X  -127.452, Y  +285.790, Z    +0.000, E1  +303.409, E3 -64813.783}
SPL {X  -148.001, Y  +321.733, Z    +0.000, E1  +312.190, E3 -64827.887}
SPL {X  -154.604, Y  +341.337, Z    +0.000, E1  +321.370, E3 -64831.660}
SPL {X  -158.135, Y  +358.205, Z    +0.000, E1  +333.016, E3 -64833.610}
SPL {X  -159.602, Y  +371.361, Z    +0.000, E1  +345.165, E3 -64834.506}
SPL {X  -159.981, Y  +380.818, Z    +0.000, E1  +355.488, E3 -64834.784}
SPL {X  -159.990, Y  +384.681, Z    +0.000, E1  +360.222, E3 -64834.813}
SPL {X  -159.990, Y  +387.626, Z    +0.000, E1  +368.190, E3 -64834.841}
SPL {X  -159.990, Y  +390.340, Z    +0.000, E1  +375.987, E3 -64834.906}
SPL {X  -159.990, Y  +394.216, Z    +0.000, E1  +387.062, E3 -64835.068}
SPL {X  -159.990, Y  +399.855, Z    +0.000, E1  +400.916, E3 -64835.439}
SPL {X  -159.990, Y  +405.475, Z    +0.000, E1  +411.039, E3 -64835.956}
SPL {X  -159.990, Y  +414.231, Z    +0.000, E1  +420.575, E3 -64837.140}
SPL {X  -159.990, Y  +462.953, Z    +0.000, E1  +433.611, E3 -64848.879}
SPL {X  -153.839, Y  +715.436, Z    +0.000, E1  +435.884, E3 -64951.310}
SPL {X  -149.923, Y  +727.355, Z    +0.000, E1  +435.515, E3 -64961.419}
SPL {X  -145.995, Y  +736.939, Z    +0.000, E1  +435.150, E3 -64970.154}
SPL {X  -141.012, Y  +747.080, Z    +0.000, E1  +434.661, E3 -64980.006}
SPL {X  -136.371, Y  +755.165, Z    +0.000, E1  +434.152, E3 -64988.292}
SPL {X  -131.455, Y  +762.694, Z    +0.000, E1  +433.615, E3 -64996.210}
SPL {X  -125.933, Y  +770.180, Z    +0.000, E1  +432.934, E3 -65004.275}
SPL {X  -121.698, Y  +775.357, Z    +0.000, E1  +432.353, E3 -65009.840}
SPL {X  -118.622, Y  +778.858, Z    +0.000, E1  +431.924, E3 -65013.466}
SPL {X   -66.171, Y  +817.165, Z    +0.000, E1  +416.016, E3 -65164.824}
ENDSPLINE

SPLINE
SPL {X  -126.418, Y  +769.557, Z    +0.000, E1  +417.118, E3 -65348.065}
SPL {X  -148.476, Y  +731.097, Z    +0.000, E1  +407.824, E3 -65363.221}
SPL {X  -156.642, Y  +704.059, Z    +0.000, E1  +393.659, E3 -65367.863}
SPL {X  -159.317, Y  +686.157, Z    +0.000, E1  +378.660, E3 -65369.353}
SPL {X  -159.973, Y  +673.799, Z    +0.000, E1  +365.345, E3 -65369.802}
SPL {X  -159.990, Y  +669.500, Z    +0.000, E1  +360.000, E3 -65369.842}
SPL {X  -159.990, Y  +667.794, Z    +0.000, E1  +355.745, E3 -65369.853}
SPL {X  -159.990, Y  +664.091, Z    +0.000, E1  +345.072, E3 -65369.925}
SPL {X  -159.990, Y  +659.599, Z    +0.000, E1  +331.984, E3 -65370.096}
SPL {X  -159.990, Y  +652.711, Z    +0.000, E1  +315.707, E3 -65370.575}
SPL {X  -159.990, Y  +640.730, Z    +0.000, E1  +299.703, E3 -65371.924}
SPL {X  -159.990, Y  +620.478, Z    +0.000, E1  +289.974, E3 -65375.738}
SPL {X  -159.990, Y  +573.021, Z    +0.000, E1  +285.381, E3 -65389.681}
SPL {X  -154.165, Y  +339.724, Z    +0.000, E1  +284.073, E3 -65485.528}
SPL {X  -150.223, Y  +327.456, Z    +0.000, E1  +284.427, E3 -65495.793}
SPL {X  -136.549, Y  +299.126, Z    +0.000, E1  +282.463, E3 -65488.683}
ENDSPLINE

SPLINE
SPL {X  -136.862, Y  +299.641, Z    +0.000, E1  +283.396, E3 -65497.325}
ENDSPLINE

SPLINE
SPL {X  -136.434, Y  +298.938, Z    +0.000, E1  +284.018, E3 -65503.216}
SPL {X  -135.890, Y  +298.057, Z    +0.000, E1  +284.960, E3 -65511.682}
SPL {X  -134.349, Y  +295.626, Z    +0.000, E1  +285.678, E3 -65518.530}
SPL {X  -131.287, Y  +291.064, Z    +0.000, E1  +286.028, E3 -65523.342}
SPL {X  -128.265, Y  +286.871, Z    +0.000, E1  +286.387, E3 -65527.798}
SPL {X  -125.161, Y  +282.843, Z    +0.000, E1  +286.768, E3 -65532.070}
SPL {X  -122.038, Y  +279.042, Z    +0.000, E1  +287.168, E3 -65536.050}
SPL {X  -119.499, Y  +276.120, Z    +0.000, E1  +287.518, E3 -65539.069}
SPL {X  -117.726, Y  +274.160, Z    +0.000, E1  +287.766, E3 -65541.032}
SPL {X   -66.040, Y  +236.776, Z    +0.000, E1  +304.306, E3 -65701.376}
ENDSPLINE

SPLINE
SPL {X  -127.452, Y  +285.790, Z    +0.000, E1  +303.409, E3 -65875.322}
SPL {X  -148.001, Y  +321.733, Z    +0.000, E1  +312.190, E3 -65889.425}
SPL {X  -154.604, Y  +341.337, Z    +0.000, E1  +321.370, E3 -65893.199}
SPL {X  -158.135, Y  +358.205, Z    +0.000, E1  +333.016, E3 -65895.149}
SPL {X  -159.602, Y  +371.361, Z    +0.000, E1  +345.165, E3 -65896.045}
SPL {X  -159.981, Y  +380.818, Z    +0.000, E1  +355.488, E3 -65896.322}
SPL {X  -159.990, Y  +384.681, Z    +0.000, E1  +360.222, E3 -65896.351}
SPL {X  -159.990, Y  +387.626, Z    +0.000, E1  +368.190, E3 -65896.380}
SPL {X  -159.990, Y  +390.340, Z    +0.000, E1  +375.987, E3 -65896.444}
SPL {X  -159.990, Y  +394.216, Z    +0.000, E1  +387.062, E3 -65896.606}
SPL {X  -159.990, Y  +399.855, Z    +0.000, E1  +400.916, E3 -65896.977}
SPL {X  -159.990, Y  +405.475, Z    +0.000, E1  +411.039, E3 -65897.494}
SPL {X  -159.990, Y  +414.231, Z    +0.000, E1  +420.575, E3 -65898.678}
SPL {X  -159.990, Y  +462.953, Z    +0.000, E1  +433.611, E3 -65910.417}
SPL {X  -153.839, Y  +715.436, Z    +0.000, E1  +435.884, E3 -66012.848}
SPL {X  -148.840, Y  +730.182, Z    +0.000, E1  +435.434, E3 -66025.425}
SPL {X  -143.409, Y  +742.426, Z    +0.000, E1  +434.905, E3 -66036.937}
SPL {X  -139.557, Y  +749.735, Z    +0.000, E1  +434.483, E3 -66044.285}
SPL {X  -136.371, Y  +755.165, Z    +0.000, E1  +434.152, E3 -66049.830}
SPL {X  -131.455, Y  +762.694, Z    +0.000, E1  +433.615, E3 -66057.748}
SPL {X  -125.933, Y  +770.180, Z    +0.000, E1  +432.934, E3 -66065.813}
SPL {X  -121.698, Y  +775.357, Z    +0.000, E1  +432.353, E3 -66071.378}
SPL {X  -118.622, Y  +778.858, Z    +0.000, E1  +431.924, E3 -66075.004}
SPL {X   -66.171, Y  +817.165, Z    +0.000, E1  +416.016, E3 -66226.363}
ENDSPLINE

SPLINE
SPL {X  -126.418, Y  +769.557, Z    +0.000, E1  +417.118, E3 -66409.604}
SPL {X  -145.244, Y  +738.589, Z    +0.000, E1  +410.405, E3 -66422.845}
SPL {X  -150.151, Y  +726.741, Z    +0.000, E1  +406.068, E3 -66425.772}
SPL {X  -156.642, Y  +704.059, Z    +0.000, E1  +393.659, E3 -66429.402}
SPL {X  -159.317, Y  +686.157, Z    +0.000, E1  +378.660, E3 -66430.892}
SPL {X  -159.973, Y  +673.799, Z    +0.000, E1  +365.345, E3 -66431.340}
SPL {X  -159.990, Y  +669.500, Z    +0.000, E1  +360.000, E3 -66431.381}
SPL {X  -159.990, Y  +667.794, Z    +0.000, E1  +355.745, E3 -66431.392}
SPL {X  -159.990, Y  +664.091, Z    +0.000, E1  +345.072, E3 -66431.464}
SPL {X  -159.990, Y  +659.599, Z    +0.000, E1  +331.984, E3 -66431.634}
SPL {X  -159.990, Y  +652.711, Z    +0.000, E1  +315.707, E3 -66432.114}
SPL {X  -159.990, Y  +640.730, Z    +0.000, E1  +299.703, E3 -66433.463}
SPL {X  -159.990, Y  +620.478, Z    +0.000, E1  +289.974, E3 -66437.276}
SPL {X  -159.990, Y  +573.021, Z    +0.000, E1  +285.381, E3 -66451.220}
SPL {X  -154.165, Y  +339.724, Z    +0.000, E1  +284.073, E3 -66547.067}
SPL {X  -150.223, Y  +327.456, Z    +0.000, E1  +284.427, E3 -66557.332}
SPL {X  -136.549, Y  +299.126, Z    +0.000, E1  +282.463, E3 -66550.222}
ENDSPLINE

SPLINE
SPL {X  -136.626, Y  +299.252, Z    +0.000, E1  +283.686, E3 -66561.872}
ENDSPLINE

SPLINE
SPL {X  -135.890, Y  +298.057, Z    +0.000, E1  +284.960, E3 -66573.221}
SPL {X  -134.349, Y  +295.626, Z    +0.000, E1  +285.678, E3 -66580.068}
SPL {X  -131.287, Y  +291.064, Z    +0.000, E1  +286.028, E3 -66584.881}
SPL {X  -128.265, Y  +286.871, Z    +0.000, E1  +286.387, E3 -66589.337}
SPL {X  -125.161, Y  +282.843, Z    +0.000, E1  +286.768, E3 -66593.608}
SPL {X  -122.038, Y  +279.042, Z    +0.000, E1  +287.168, E3 -66597.588}
SPL {X  -118.642, Y  +275.165, Z    +0.000, E1  +287.619, E3 -66601.551}
SPL {X   -66.040, Y  +236.776, Z    +0.000, E1  +304.306, E3 -66762.915}
ENDSPLINE

SPLINE
SPL {X  -127.452, Y  +285.790, Z    +0.000, E1  +303.409, E3 -66936.860}
SPL {X  -151.591, Y  +331.344, Z    +0.000, E1  +316.130, E3 -66952.959}
SPL {X  -158.135, Y  +358.205, Z    +0.000, E1  +333.016, E3 -66956.687}
SPL {X  -159.602, Y  +371.361, Z    +0.000, E1  +345.165, E3 -66957.583}
SPL {X  -159.981, Y  +380.818, Z    +0.000, E1  +355.488, E3 -66957.861}
SPL {X  -159.990, Y  +384.681, Z    +0.000, E1  +360.222, E3 -66957.890}
SPL {X  -159.990, Y  +389.079, Z    +0.000, E1  +372.017, E3 -66957.953}
SPL {X  -159.990, Y  +394.216, Z    +0.000, E1  +387.062, E3 -66958.145}
SPL {X  -159.990, Y  +401.720, Z    +0.000, E1  +404.434, E3 -66958.687}
SPL {X  -159.990, Y  +414.231, Z    +0.000, E1  +420.575, E3 -66960.217}
SPL {X  -159.990, Y  +462.953, Z    +0.000, E1  +433.611, E3 -66971.956}
SPL {X  -155.068, Y  +710.881, Z    +0.000, E1  +435.973, E3 -67070.842}
SPL {X  -152.790, Y  +718.955, Z    +0.000, E1  +435.770, E3 -67077.327}
SPL {X  -148.840, Y  +730.182, Z    +0.000, E1  +435.434, E3 -67086.963}
SPL {X  -143.409, Y  +742.426, Z    +0.000, E1  +434.905, E3 -67098.475}
SPL {X  -139.557, Y  +749.735, Z    +0.000, E1  +434.483, E3 -67105.823}
SPL {X  -136.371, Y  +755.165, Z    +0.000, E1  +434.152, E3 -67111.369}
SPL {X  -133.102, Y  +760.274, Z    +0.000, E1  +433.777, E3 -67116.754}
SPL {X  -128.975, Y  +766.169, Z    +0.000, E1  +433.313, E3 -67123.029}
SPL {X  -124.947, Y  +771.425, Z    +0.000, E1  +432.782, E3 -67128.722}
SPL {X  -121.698, Y  +775.357, Z    +0.000, E1  +432.353, E3 -67132.917}
SPL {X  -118.622, Y  +778.858, Z    +0.000, E1  +431.924, E3 -67136.543}
SPL {X   -66.171, Y  +817.165, Z    +0.000, E1  +416.016, E3 -67287.901}
ENDSPLINE

SPLINE
SPL {X  -126.418, Y  +769.557, Z    +0.000, E1  +417.118, E3 -67471.142}
SPL {X  -145.244, Y  +738.589, Z    +0.000, E1  +410.405, E3 -67484.384}
SPL {X  -150.151, Y  +726.741, Z    +0.000, E1  +406.068, E3 -67487.311}
SPL {X  -156.642, Y  +704.059, Z    +0.000, E1  +393.659, E3 -67490.940}
SPL {X  -159.317, Y  +686.157, Z    +0.000, E1  +378.660, E3 -67492.430}
SPL {X  -159.907, Y  +676.666, Z    +0.000, E1  +368.555, E3 -67492.828}
SPL {X  -159.990, Y  +669.586, Z    +0.000, E1  +360.216, E3 -67492.919}
SPL {X  -159.990, Y  +667.794, Z    +0.000, E1  +355.745, E3 -67492.930}
SPL {X  -159.990, Y  +664.091, Z    +0.000, E1  +345.072, E3 -67493.002}
SPL {X  -159.990, Y  +659.599, Z    +0.000, E1  +331.984, E3 -67493.173}
SPL {X  -159.990, Y  +652.711, Z    +0.000, E1  +315.707, E3 -67493.652}
SPL {X  -159.990, Y  +640.730, Z    +0.000, E1  +299.703, E3 -67495.001}
SPL {X  -159.990, Y  +620.478, Z    +0.000, E1  +289.974, E3 -67498.814}
SPL {X  -159.990, Y  +573.021, Z    +0.000, E1  +285.381, E3 -67512.758}
SPL {X  -154.165, Y  +339.724, Z    +0.000, E1  +284.073, E3 -67608.605}
SPL {X  -150.223, Y  +327.456, Z    +0.000, E1  +284.427, E3 -67618.870}
SPL {X  -136.549, Y  +299.126, Z    +0.000, E1  +282.463, E3 -67611.760}
ENDSPLINE

SPLINE
SPL {X  -136.626, Y  +299.252, Z    +0.000, E1  +283.686, E3 -67623.410}
ENDSPLINE

SPLINE
SPL {X  -135.890, Y  +298.057, Z    +0.000, E1  +284.960, E3 -67634.759}
SPL {X  -134.349, Y  +295.626, Z    +0.000, E1  +285.678, E3 -67641.606}
SPL {X  -131.287, Y  +291.064, Z    +0.000, E1  +286.028, E3 -67646.419}
SPL {X  -128.265, Y  +286.871, Z    +0.000, E1  +286.387, E3 -67650.875}
SPL {X  -125.161, Y  +282.843, Z    +0.000, E1  +286.768, E3 -67655.147}
SPL {X  -122.038, Y  +279.042, Z    +0.000, E1  +287.168, E3 -67659.127}
SPL {X  -119.499, Y  +276.120, Z    +0.000, E1  +287.518, E3 -67662.146}
SPL {X  -117.726, Y  +274.160, Z    +0.000, E1  +287.766, E3 -67664.109}
SPL {X   -66.040, Y  +236.776, Z    +0.000, E1  +304.306, E3 -67824.453}
ENDSPLINE

SPLINE
SPL {X  -127.452, Y  +285.790, Z    +0.000, E1  +303.409, E3 -67998.399}
SPL {X  -151.591, Y  +331.344, Z    +0.000, E1  +316.130, E3 -68014.498}
SPL {X  -158.135, Y  +358.205, Z    +0.000, E1  +333.016, E3 -68018.226}
SPL {X  -159.602, Y  +371.361, Z    +0.000, E1  +345.165, E3 -68019.122}
SPL {X  -159.981, Y  +380.818, Z    +0.000, E1  +355.488, E3 -68019.399}
SPL {X  -159.990, Y  +384.681, Z    +0.000, E1  +360.222, E3 -68019.428}
SPL {X  -159.990, Y  +387.626, Z    +0.000, E1  +368.190, E3 -68019.457}
SPL {X  -159.990, Y  +390.340, Z    +0.000, E1  +375.987, E3 -68019.521}
SPL {X  -159.990, Y  +394.216, Z    +0.000, E1  +387.062, E3 -68019.683}
SPL {X  -159.990, Y  +399.855, Z    +0.000, E1  +400.916, E3 -68020.054}
SPL {X  -159.990, Y  +405.475, Z    +0.000, E1  +411.039, E3 -68020.571}
SPL {X  -159.990, Y  +414.231, Z    +0.000, E1  +420.575, E3 -68021.755}
SPL {X  -159.990, Y  +462.953, Z    +0.000, E1  +433.611, E3 -68033.494}
SPL {X  -153.839, Y  +715.436, Z    +0.000, E1  +435.884, E3 -68135.925}
SPL {X  -148.840, Y  +730.182, Z    +0.000, E1  +435.434, E3 -68148.502}
SPL {X  -143.409, Y  +742.426, Z    +0.000, E1  +434.905, E3 -68160.014}
SPL {X  -139.557, Y  +749.735, Z    +0.000, E1  +434.483, E3 -68167.362}
SPL {X  -136.371, Y  +755.165, Z    +0.000, E1  +434.152, E3 -68172.907}
SPL {X  -133.102, Y  +760.274, Z    +0.000, E1  +433.777, E3 -68178.292}
SPL {X  -128.975, Y  +766.169, Z    +0.000, E1  +433.313, E3 -68184.568}
SPL {X  -124.947, Y  +771.425, Z    +0.000, E1  +432.782, E3 -68190.261}
SPL {X  -121.698, Y  +775.357, Z    +0.000, E1  +432.353, E3 -68194.455}
SPL {X  -118.622, Y  +778.858, Z    +0.000, E1  +431.924, E3 -68198.081}
SPL {X   -66.171, Y  +817.165, Z    +0.000, E1  +416.016, E3 -68349.440}
ENDSPLINE

SPLINE
SPL {X  -126.418, Y  +769.557, Z    +0.000, E1  +417.118, E3 -68532.681}
SPL {X  -145.244, Y  +738.589, Z    +0.000, E1  +410.405, E3 -68545.922}
SPL {X  -150.151, Y  +726.741, Z    +0.000, E1  +406.068, E3 -68548.849}
SPL {X  -156.642, Y  +704.059, Z    +0.000, E1  +393.659, E3 -68552.479}
SPL {X  -159.317, Y  +686.157, Z    +0.000, E1  +378.660, E3 -68553.969}
SPL {X  -159.973, Y  +673.799, Z    +0.000, E1  +365.345, E3 -68554.417}
SPL {X  -159.990, Y  +669.500, Z    +0.000, E1  +360.000, E3 -68554.457}
SPL {X  -159.990, Y  +667.794, Z    +0.000, E1  +355.745, E3 -68554.469}
SPL {X  -159.990, Y  +664.091, Z    +0.000, E1  +345.072, E3 -68554.541}
SPL {X  -159.990, Y  +659.599, Z    +0.000, E1  +331.984, E3 -68554.711}
SPL {X  -159.990, Y  +652.711, Z    +0.000, E1  +315.707, E3 -68555.191}
SPL {X  -159.990, Y  +640.730, Z    +0.000, E1  +299.703, E3 -68556.540}
SPL {X  -159.990, Y  +620.478, Z    +0.000, E1  +289.974, E3 -68560.353}
SPL {X  -159.990, Y  +573.021, Z    +0.000, E1  +285.381, E3 -68574.297}
SPL {X  -154.165, Y  +339.724, Z    +0.000, E1  +284.073, E3 -68670.144}
SPL {X  -150.571, Y  +328.416, Z    +0.000, E1  +284.401, E3 -68679.589}
SPL {X  -148.206, Y  +322.236, Z    +0.000, E1  +284.635, E3 -68685.133}
SPL {X  -136.549, Y  +299.126, Z    +0.000, E1  +282.463, E3 -68673.299}
ENDSPLINE

SPLINE
SPL {X  -136.862, Y  +299.641, Z    +0.000, E1  +283.396, E3 -68681.941}
ENDSPLINE

SPLINE
SPL {X  -136.434, Y  +298.938, Z    +0.000, E1  +284.018, E3 -68687.832}
SPL {X  -135.838, Y  +297.973, Z    +0.000, E1  +284.965, E3 -68696.380}
ENDSPLINE

SPLINE
SPL {X  -138.785, Y  +302.903, Z    +0.000, E1  +287.056, E3 -68710.413}
ENDSPLINE

SPLINE
SPL {X  -135.531, Y  +297.482, Z    +0.000, E1  +287.444, E3 -68716.329}
SPL {X  -132.271, Y  +292.493, Z    +0.000, E1  +287.844, E3 -68721.847}
SPL {X  -128.837, Y  +287.643, Z    +0.000, E1  +288.283, E3 -68727.285}
SPL {X  -124.965, Y  +282.598, Z    +0.000, E1  +288.800, E3 -68732.946}
SPL {X  -120.791, Y  +277.589, Z    +0.000, E1  +289.397, E3 -68738.519}
SPL {X   -74.058, Y  +240.683, Z    +0.000, E1  +305.011, E3 -68895.582}
ENDSPLINE

SPLINE
SPL {X  -130.401, Y  +289.805, Z    +0.000, E1  +307.505, E3 -69052.553}
SPL {X  -148.502, Y  +322.968, Z    +0.000, E1  +316.497, E3 -69066.873}
SPL {X  -154.800, Y  +342.080, Z    +0.000, E1  +325.471, E3 -69071.177}
SPL {X  -158.218, Y  +358.753, Z    +0.000, E1  +336.397, E3 -69073.537}
SPL {X  -159.681, Y  +372.564, Z    +0.000, E1  +347.981, E3 -69074.589}
SPL {X  -159.987, Y  +381.561, Z    +0.000, E1  +356.806, E3 -69074.885}
SPL {X  -159.990, Y  +384.668, Z    +0.000, E1  +360.183, E3 -69074.911}
SPL {X  -159.990, Y  +387.837, Z    +0.000, E1  +367.342, E3 -69074.951}
SPL {X  -159.990, Y  +393.084, Z    +0.000, E1  +380.137, E3 -69075.161}
SPL {X  -159.990, Y  +401.914, Z    +0.000, E1  +400.147, E3 -69075.855}
SPL {X  -159.990, Y  +414.609, Z    +0.000, E1  +416.791, E3 -69077.592}
SPL {X  -159.990, Y  +464.476, Z    +0.000, E1  +431.765, E3 -69090.393}
SPL {X  -157.643, Y  +698.802, Z    +0.000, E1  +434.751, E3 -69193.407}
SPL {X  -154.470, Y  +713.164, Z    +0.000, E1  +434.425, E3 -69204.996}
SPL {X  -151.032, Y  +724.285, Z    +0.000, E1  +434.102, E3 -69214.800}
SPL {X  -147.134, Y  +734.337, Z    +0.000, E1  +433.686, E3 -69224.437}
SPL {X  -143.804, Y  +741.622, Z    +0.000, E1  +433.324, E3 -69231.825}
SPL {X  -140.603, Y  +747.839, Z    +0.000, E1  +432.964, E3 -69238.341}
SPL {X  -137.184, Y  +753.824, Z    +0.000, E1  +432.574, E3 -69244.778}
SPL {X  -133.762, Y  +759.276, Z    +0.000, E1  +432.150, E3 -69250.831}
SPL {X  -130.927, Y  +763.451, Z    +0.000, E1  +431.785, E3 -69255.526}
SPL {X  -128.105, Y  +767.343, Z    +0.000, E1  +431.419, E3 -69259.915}
SPL {X  -124.554, Y  +771.914, Z    +0.000, E1  +430.935, E3 -69265.086}
SPL {X  -120.892, Y  +776.295, Z    +0.000, E1  +430.404, E3 -69269.969}
SPL {X  -118.039, Y  +779.498, Z    +0.000, E1  +429.949, E3 -69273.487}
SPL {X   -71.924, Y  +814.412, Z    +0.000, E1  +415.124, E3 -69428.243}
ENDSPLINE

SPLINE
SPL {X  -132.255, Y  +761.530, Z    +0.000, E1  +413.203, E3 -69591.413}
SPL {X  -150.415, Y  +726.018, Z    +0.000, E1  +402.769, E3 -69604.917}
SPL {X  -156.153, Y  +706.328, Z    +0.000, E1  +392.414, E3 -69608.609}
SPL {X  -159.178, Y  +687.603, Z    +0.000, E1  +378.267, E3 -69610.587}
SPL {X  -159.974, Y  +673.783, Z    +0.000, E1  +364.843, E3 -69611.209}
SPL {X  -159.990, Y  +669.500, Z    +0.000, E1  +360.000, E3 -69611.256}
SPL {X  -159.990, Y  +667.470, Z    +0.000, E1  +355.588, E3 -69611.274}
SPL {X  -159.990, Y  +662.995, Z    +0.000, E1  +343.976, E3 -69611.391}
SPL {X  -159.990, Y  +658.179, Z    +0.000, E1  +331.312, E3 -69611.628}
SPL {X  -159.990, Y  +652.822, Z    +0.000, E1  +319.345, E3 -69612.042}
SPL {X  -159.990, Y  +646.185, Z    +0.000, E1  +308.728, E3 -69612.781}
SPL {X  -159.990, Y  +636.375, Z    +0.000, E1  +299.286, E3 -69614.220}
SPL {X  -159.990, Y  +617.374, Z    +0.000, E1  +291.478, E3 -69618.547}
SPL {X  -159.990, Y  +579.000, Z    +0.000, E1  +286.931, E3 -69630.006}
SPL {X  -157.725, Y  +355.675, Z    +0.000, E1  +284.959, E3 -69726.964}
SPL {X  -142.593, Y  +309.947, Z    +0.000, E1  +282.426, E3 -69720.628}
SPL {X  -142.198, Y  +309.176, Z    +0.000, E1  +283.218, E3 -69729.436}
ENDSPLINE

SPLINE
SPL {X  -142.352, Y  +309.474, Z    +0.000, E1  +284.206, E3 -69739.130}
ENDSPLINE

SPLINE
SPL {X  -141.553, Y  +307.937, Z    +0.000, E1  +285.290, E3 -69750.146}
SPL {X  -140.562, Y  +306.086, Z    +0.000, E1  +286.440, E3 -69760.839}
SPL {X  -138.743, Y  +302.832, Z    +0.000, E1  +287.062, E3 -69767.637}
SPL {X  -135.531, Y  +297.482, Z    +0.000, E1  +287.444, E3 -69773.471}
SPL {X  -132.271, Y  +292.493, Z    +0.000, E1  +287.844, E3 -69778.990}
SPL {X  -128.837, Y  +287.643, Z    +0.000, E1  +288.283, E3 -69784.428}
SPL {X  -124.965, Y  +282.598, Z    +0.000, E1  +288.800, E3 -69790.089}
SPL {X  -120.791, Y  +277.589, Z    +0.000, E1  +289.397, E3 -69795.662}
SPL {X   -74.058, Y  +240.683, Z    +0.000, E1  +305.011, E3 -69952.725}
ENDSPLINE

SPLINE
SPL {X  -130.401, Y  +289.805, Z    +0.000, E1  +307.505, E3 -70109.696}
SPL {X  -148.502, Y  +322.968, Z    +0.000, E1  +316.497, E3 -70124.016}
SPL {X  -154.800, Y  +342.080, Z    +0.000, E1  +325.471, E3 -70128.320}
SPL {X  -158.218, Y  +358.753, Z    +0.000, E1  +336.397, E3 -70130.680}
SPL {X  -159.681, Y  +372.564, Z    +0.000, E1  +347.981, E3 -70131.731}
SPL {X  -159.987, Y  +381.561, Z    +0.000, E1  +356.806, E3 -70132.028}
SPL {X  -159.990, Y  +384.668, Z    +0.000, E1  +360.183, E3 -70132.054}
SPL {X  -159.990, Y  +387.837, Z    +0.000, E1  +367.342, E3 -70132.094}
SPL {X  -159.990, Y  +393.084, Z    +0.000, E1  +380.137, E3 -70132.304}
SPL {X  -159.990, Y  +401.914, Z    +0.000, E1  +400.147, E3 -70132.998}
SPL {X  -159.990, Y  +414.609, Z    +0.000, E1  +416.791, E3 -70134.735}
SPL {X  -159.990, Y  +464.476, Z    +0.000, E1  +431.765, E3 -70147.536}
SPL {X  -157.643, Y  +698.802, Z    +0.000, E1  +434.751, E3 -70250.550}
SPL {X  -154.470, Y  +713.164, Z    +0.000, E1  +434.425, E3 -70262.139}
SPL {X  -151.032, Y  +724.285, Z    +0.000, E1  +434.102, E3 -70271.943}
SPL {X  -147.134, Y  +734.337, Z    +0.000, E1  +433.686, E3 -70281.580}
SPL {X  -143.804, Y  +741.622, Z    +0.000, E1  +433.324, E3 -70288.968}
SPL {X  -140.603, Y  +747.839, Z    +0.000, E1  +432.964, E3 -70295.484}
SPL {X  -137.184, Y  +753.824, Z    +0.000, E1  +432.574, E3 -70301.920}
SPL {X  -133.762, Y  +759.276, Z    +0.000, E1  +432.150, E3 -70307.974}
SPL {X  -130.927, Y  +763.451, Z    +0.000, E1  +431.785, E3 -70312.669}
SPL {X  -128.105, Y  +767.343, Z    +0.000, E1  +431.419, E3 -70317.058}
SPL {X  -124.554, Y  +771.914, Z    +0.000, E1  +430.935, E3 -70322.229}
SPL {X  -120.892, Y  +776.295, Z    +0.000, E1  +430.404, E3 -70327.112}
SPL {X  -118.039, Y  +779.498, Z    +0.000, E1  +429.949, E3 -70330.630}
SPL {X   -71.966, Y  +814.391, Z    +0.000, E1  +415.783, E3 -70469.283}
ENDSPLINE

SPLINE
SPL {X  -117.449, Y  +780.140, Z    +0.000, E1  +415.491, E3 -70633.697}
SPL {X  -137.837, Y  +752.727, Z    +0.000, E1  +411.385, E3 -70653.185}
SPL {X  -150.415, Y  +726.018, Z    +0.000, E1  +402.769, E3 -70662.060}
SPL {X  -156.153, Y  +706.328, Z    +0.000, E1  +392.414, E3 -70665.752}
SPL {X  -159.178, Y  +687.603, Z    +0.000, E1  +378.267, E3 -70667.730}
SPL {X  -159.915, Y  +676.399, Z    +0.000, E1  +367.484, E3 -70668.300}
SPL {X  -159.990, Y  +669.381, Z    +0.000, E1  +359.965, E3 -70668.400}
SPL {X  -159.990, Y  +666.412, Z    +0.000, E1  +352.765, E3 -70668.431}
SPL {X  -159.990, Y  +662.995, Z    +0.000, E1  +343.976, E3 -70668.534}
SPL {X  -159.990, Y  +658.179, Z    +0.000, E1  +331.312, E3 -70668.770}
SPL {X  -159.990, Y  +652.822, Z    +0.000, E1  +319.345, E3 -70669.185}
SPL {X  -159.990, Y  +646.185, Z    +0.000, E1  +308.728, E3 -70669.924}
SPL {X  -159.990, Y  +632.371, Z    +0.000, E1  +297.040, E3 -70672.276}
SPL {X  -159.990, Y  +579.000, Z    +0.000, E1  +286.931, E3 -70687.149}
SPL {X  -157.725, Y  +355.675, Z    +0.000, E1  +284.959, E3 -70784.107}
SPL {X  -142.593, Y  +309.947, Z    +0.000, E1  +282.426, E3 -70777.770}
SPL {X  -142.198, Y  +309.176, Z    +0.000, E1  +283.218, E3 -70786.579}
ENDSPLINE

SPLINE
SPL {X  -142.352, Y  +309.474, Z    +0.000, E1  +284.206, E3 -70796.273}
ENDSPLINE

SPLINE
SPL {X  -141.553, Y  +307.937, Z    +0.000, E1  +285.290, E3 -70807.288}
SPL {X  -140.562, Y  +306.086, Z    +0.000, E1  +286.440, E3 -70817.982}
SPL {X  -138.743, Y  +302.832, Z    +0.000, E1  +287.062, E3 -70824.780}
SPL {X  -135.531, Y  +297.482, Z    +0.000, E1  +287.444, E3 -70830.614}
SPL {X  -132.271, Y  +292.493, Z    +0.000, E1  +287.844, E3 -70836.133}
SPL {X  -128.837, Y  +287.643, Z    +0.000, E1  +288.283, E3 -70841.570}
SPL {X  -125.941, Y  +283.830, Z    +0.000, E1  +288.683, E3 -70845.870}
SPL {X  -122.669, Y  +279.791, Z    +0.000, E1  +289.119, E3 -70850.364}
SPL {X  -119.730, Y  +276.380, Z    +0.000, E1  +289.584, E3 -70854.152}
SPL {X   -74.058, Y  +240.683, Z    +0.000, E1  +305.011, E3 -71009.868}
ENDSPLINE

SPLINE
SPL {X  -130.401, Y  +289.805, Z    +0.000, E1  +307.505, E3 -71166.839}
SPL {X  -148.502, Y  +322.968, Z    +0.000, E1  +316.497, E3 -71181.159}
SPL {X  -154.800, Y  +342.080, Z    +0.000, E1  +325.471, E3 -71185.463}
SPL {X  -158.218, Y  +358.753, Z    +0.000, E1  +336.397, E3 -71187.823}
SPL {X  -159.681, Y  +372.564, Z    +0.000, E1  +347.981, E3 -71188.874}
SPL {X  -159.987, Y  +381.561, Z    +0.000, E1  +356.806, E3 -71189.171}
SPL {X  -159.990, Y  +384.668, Z    +0.000, E1  +360.183, E3 -71189.196}
SPL {X  -159.990, Y  +387.837, Z    +0.000, E1  +367.342, E3 -71189.237}
SPL {X  -159.990, Y  +393.084, Z    +0.000, E1  +380.137, E3 -71189.447}
SPL {X  -159.990, Y  +401.914, Z    +0.000, E1  +400.147, E3 -71190.141}
SPL {X  -159.990, Y  +414.609, Z    +0.000, E1  +416.791, E3 -71191.877}
SPL {X  -159.990, Y  +464.476, Z    +0.000, E1  +431.765, E3 -71204.678}
SPL {X  -157.643, Y  +698.802, Z    +0.000, E1  +434.751, E3 -71307.693}
SPL {X  -154.470, Y  +713.164, Z    +0.000, E1  +434.425, E3 -71319.282}
SPL {X  -151.032, Y  +724.285, Z    +0.000, E1  +434.102, E3 -71329.086}
SPL {X  -147.134, Y  +734.337, Z    +0.000, E1  +433.686, E3 -71338.723}
SPL {X  -143.804, Y  +741.622, Z    +0.000, E1  +433.324, E3 -71346.111}
SPL {X  -140.603, Y  +747.839, Z    +0.000, E1  +432.964, E3 -71352.627}
SPL {X  -137.184, Y  +753.824, Z    +0.000, E1  +432.574, E3 -71359.063}
SPL {X  -133.762, Y  +759.276, Z    +0.000, E1  +432.150, E3 -71365.117}
SPL {X  -130.927, Y  +763.451, Z    +0.000, E1  +431.785, E3 -71369.812}
SPL {X  -128.105, Y  +767.343, Z    +0.000, E1  +431.419, E3 -71374.200}
SPL {X  -124.554, Y  +771.914, Z    +0.000, E1  +430.935, E3 -71379.371}
SPL {X  -120.892, Y  +776.295, Z    +0.000, E1  +430.404, E3 -71384.255}
SPL {X  -118.039, Y  +779.498, Z    +0.000, E1  +429.949, E3 -71387.773}
SPL {X   -71.966, Y  +814.391, Z    +0.000, E1  +415.783, E3 -71526.425}
ENDSPLINE

SPLINE
SPL {X  -117.449, Y  +780.140, Z    +0.000, E1  +415.491, E3 -71690.840}
SPL {X  -137.837, Y  +752.727, Z    +0.000, E1  +411.385, E3 -71710.328}
SPL {X  -150.415, Y  +726.018, Z    +0.000, E1  +402.769, E3 -71719.203}
SPL {X  -156.153, Y  +706.328, Z    +0.000, E1  +392.414, E3 -71722.895}
SPL {X  -159.178, Y  +687.603, Z    +0.000, E1  +378.267, E3 -71724.873}
SPL {X  -159.915, Y  +676.399, Z    +0.000, E1  +367.484, E3 -71725.443}
SPL {X  -159.990, Y  +669.381, Z    +0.000, E1  +359.965, E3 -71725.543}
SPL {X  -159.990, Y  +666.412, Z    +0.000, E1  +352.765, E3 -71725.574}
SPL {X  -159.990, Y  +662.995, Z    +0.000, E1  +343.976, E3 -71725.677}
SPL {X  -159.990, Y  +658.179, Z    +0.000, E1  +331.312, E3 -71725.913}
SPL {X  -159.990, Y  +652.822, Z    +0.000, E1  +319.345, E3 -71726.328}
SPL {X  -159.990, Y  +646.185, Z    +0.000, E1  +308.728, E3 -71727.067}
SPL {X  -159.990, Y  +632.371, Z    +0.000, E1  +297.040, E3 -71729.419}
SPL {X  -159.990, Y  +579.000, Z    +0.000, E1  +286.931, E3 -71744.292}
SPL {X  -157.725, Y  +355.675, Z    +0.000, E1  +284.959, E3 -71841.250}
SPL {X  -142.593, Y  +309.947, Z    +0.000, E1  +282.426, E3 -71834.913}
SPL {X  -142.198, Y  +309.176, Z    +0.000, E1  +283.218, E3 -71843.722}
ENDSPLINE

SPLINE
SPL {X  -142.352, Y  +309.474, Z    +0.000, E1  +284.206, E3 -71853.415}
ENDSPLINE

SPLINE
SPL {X  -141.553, Y  +307.937, Z    +0.000, E1  +285.290, E3 -71864.431}
SPL {X  -140.562, Y  +306.086, Z    +0.000, E1  +286.440, E3 -71875.125}
SPL {X  -138.743, Y  +302.832, Z    +0.000, E1  +287.062, E3 -71881.923}
SPL {X  -135.531, Y  +297.482, Z    +0.000, E1  +287.444, E3 -71887.757}
SPL {X  -132.271, Y  +292.493, Z    +0.000, E1  +287.844, E3 -71893.276}
SPL {X  -128.837, Y  +287.643, Z    +0.000, E1  +288.283, E3 -71898.713}
SPL {X  -125.941, Y  +283.830, Z    +0.000, E1  +288.683, E3 -71903.013}
SPL {X  -122.669, Y  +279.791, Z    +0.000, E1  +289.119, E3 -71907.506}
SPL {X  -119.730, Y  +276.380, Z    +0.000, E1  +289.584, E3 -71911.295}
SPL {X   -74.058, Y  +240.683, Z    +0.000, E1  +305.011, E3 -72067.011}
ENDSPLINE

SPLINE
SPL {X  -130.401, Y  +289.805, Z    +0.000, E1  +307.505, E3 -72223.982}
SPL {X  -152.244, Y  +333.323, Z    +0.000, E1  +320.871, E3 -72240.793}
SPL {X  -158.218, Y  +358.753, Z    +0.000, E1  +336.397, E3 -72244.966}
SPL {X  -159.681, Y  +372.564, Z    +0.000, E1  +347.981, E3 -72246.017}
SPL {X  -159.987, Y  +381.561, Z    +0.000, E1  +356.806, E3 -72246.314}
SPL {X  -159.990, Y  +384.668, Z    +0.000, E1  +360.183, E3 -72246.339}
SPL {X  -159.990, Y  +387.837, Z    +0.000, E1  +367.342, E3 -72246.380}
SPL {X  -159.990, Y  +393.084, Z    +0.000, E1  +380.137, E3 -72246.590}
SPL {X  -159.990, Y  +401.914, Z    +0.000, E1  +400.147, E3 -72247.283}
SPL {X  -159.990, Y  +414.609, Z    +0.000, E1  +416.791, E3 -72249.020}
SPL {X  -159.990, Y  +464.476, Z    +0.000, E1  +431.765, E3 -72261.821}
SPL {X  -157.643, Y  +698.802, Z    +0.000, E1  +434.751, E3 -72364.836}
SPL {X  -154.470, Y  +713.164, Z    +0.000, E1  +434.425, E3 -72376.425}
SPL {X  -151.032, Y  +724.285, Z    +0.000, E1  +434.102, E3 -72386.228}
SPL {X  -147.134, Y  +734.337, Z    +0.000, E1  +433.686, E3 -72395.866}
SPL {X  -143.804, Y  +741.622, Z    +0.000, E1  +433.324, E3 -72403.254}
SPL {X  -140.603, Y  +747.839, Z    +0.000, E1  +432.964, E3 -72409.769}
SPL {X  -137.184, Y  +753.824, Z    +0.000, E1  +432.574, E3 -72416.206}
SPL {X  -133.762, Y  +759.276, Z    +0.000, E1  +432.150, E3 -72422.260}
SPL {X  -130.927, Y  +763.451, Z    +0.000, E1  +431.785, E3 -72426.954}
SPL {X  -126.852, Y  +768.996, Z    +0.000, E1  +431.276, E3 -72433.185}
SPL {X  -122.512, Y  +774.396, Z    +0.000, E1  +430.640, E3 -72439.295}
SPL {X  -119.782, Y  +777.562, Z    +0.000, E1  +430.221, E3 -72442.802}
SPL {X   -71.924, Y  +814.412, Z    +0.000, E1  +415.124, E3 -72599.672}
ENDSPLINE

SPLINE
SPL {X  -132.255, Y  +761.530, Z    +0.000, E1  +413.203, E3 -72762.842}
SPL {X  -150.415, Y  +726.018, Z    +0.000, E1  +402.769, E3 -72776.346}
SPL {X  -156.153, Y  +706.328, Z    +0.000, E1  +392.414, E3 -72780.038}
SPL {X  -159.178, Y  +687.603, Z    +0.000, E1  +378.267, E3 -72782.016}
SPL {X  -159.974, Y  +673.783, Z    +0.000, E1  +364.843, E3 -72782.637}
SPL {X  -159.990, Y  +669.500, Z    +0.000, E1  +360.000, E3 -72782.685}
SPL {X  -159.990, Y  +667.470, Z    +0.000, E1  +355.588, E3 -72782.703}
SPL {X  -159.990, Y  +662.995, Z    +0.000, E1  +343.976, E3 -72782.819}
SPL {X  -159.990, Y  +658.179, Z    +0.000, E1  +331.312, E3 -72783.056}
SPL {X  -159.990, Y  +652.822, Z    +0.000, E1  +319.345, E3 -72783.471}
SPL {X  -159.990, Y  +646.185, Z    +0.000, E1  +308.728, E3 -72784.210}
SPL {X  -159.990, Y  +632.371, Z    +0.000, E1  +297.040, E3 -72786.562}
SPL {X  -159.990, Y  +579.000, Z    +0.000, E1  +286.931, E3 -72801.434}
SPL {X  -157.725, Y  +355.675, Z    +0.000, E1  +284.959, E3 -72898.393}
SPL {X  -142.593, Y  +309.947, Z    +0.000, E1  +282.426, E3 -72892.056}
SPL {X  -142.198, Y  +309.176, Z    +0.000, E1  +283.218, E3 -72900.865}
ENDSPLINE

SPLINE
SPL {X  -142.352, Y  +309.474, Z    +0.000, E1  +284.206, E3 -72910.558}
ENDSPLINE

SPLINE
SPL {X  -141.553, Y  +307.937, Z    +0.000, E1  +285.290, E3 -72921.574}
SPL {X  -140.562, Y  +306.086, Z    +0.000, E1  +286.440, E3 -72932.268}
SPL {X  -138.743, Y  +302.832, Z    +0.000, E1  +287.062, E3 -72939.065}
SPL {X  -135.531, Y  +297.482, Z    +0.000, E1  +287.444, E3 -72944.900}
SPL {X  -132.271, Y  +292.493, Z    +0.000, E1  +287.844, E3 -72950.418}
SPL {X  -128.837, Y  +287.643, Z    +0.000, E1  +288.283, E3 -72955.856}
SPL {X  -124.965, Y  +282.598, Z    +0.000, E1  +288.800, E3 -72961.518}
SPL {X  -120.791, Y  +277.589, Z    +0.000, E1  +289.397, E3 -72967.091}
SPL {X   -74.058, Y  +240.683, Z    +0.000, E1  +305.011, E3 -73124.154}
ENDSPLINE

SPLINE
SPL {X  -130.401, Y  +289.805, Z    +0.000, E1  +307.505, E3 -73281.125}
SPL {X  -148.502, Y  +322.968, Z    +0.000, E1  +316.497, E3 -73295.445}
SPL {X  -154.800, Y  +342.080, Z    +0.000, E1  +325.471, E3 -73299.749}
SPL {X  -158.218, Y  +358.753, Z    +0.000, E1  +336.397, E3 -73302.108}
SPL {X  -159.681, Y  +372.564, Z    +0.000, E1  +347.981, E3 -73303.160}
SPL {X  -159.987, Y  +381.561, Z    +0.000, E1  +356.806, E3 -73303.456}
SPL {X  -159.990, Y  +384.668, Z    +0.000, E1  +360.183, E3 -73303.482}
SPL {X  -159.990, Y  +387.837, Z    +0.000, E1  +367.342, E3 -73303.523}
SPL {X  -159.990, Y  +393.084, Z    +0.000, E1  +380.137, E3 -73303.733}
SPL {X  -159.990, Y  +401.914, Z    +0.000, E1  +400.147, E3 -73304.426}
SPL {X  -159.990, Y  +414.609, Z    +0.000, E1  +416.791, E3 -73306.163}
SPL {X  -159.990, Y  +464.476, Z    +0.000, E1  +431.765, E3 -73318.964}
SPL {X  -157.643, Y  +698.802, Z    +0.000, E1  +434.751, E3 -73421.979}
SPL {X  -154.470, Y  +713.164, Z    +0.000, E1  +434.425, E3 -73433.568}
SPL {X  -151.032, Y  +724.285, Z    +0.000, E1  +434.102, E3 -73443.371}
SPL {X  -147.134, Y  +734.337, Z    +0.000, E1  +433.686, E3 -73453.009}
SPL {X  -143.804, Y  +741.622, Z    +0.000, E1  +433.324, E3 -73460.397}
SPL {X  -140.603, Y  +747.839, Z    +0.000, E1  +432.964, E3 -73466.912}
SPL {X  -137.184, Y  +753.824, Z    +0.000, E1  +432.574, E3 -73473.349}
SPL {X  -133.762, Y  +759.276, Z    +0.000, E1  +432.150, E3 -73479.403}
SPL {X  -130.927, Y  +763.451, Z    +0.000, E1  +431.785, E3 -73484.097}
SPL {X  -126.852, Y  +768.996, Z    +0.000, E1  +431.276, E3 -73490.328}
SPL {X  -122.512, Y  +774.396, Z    +0.000, E1  +430.640, E3 -73496.437}
SPL {X  -119.782, Y  +777.562, Z    +0.000, E1  +430.221, E3 -73499.945}
SPL {X   -71.924, Y  +814.412, Z    +0.000, E1  +415.124, E3 -73656.815}
ENDSPLINE

SPLINE
SPL {X  -132.255, Y  +761.530, Z    +0.000, E1  +413.203, E3 -73819.984}
SPL {X  -150.415, Y  +726.018, Z    +0.000, E1  +402.769, E3 -73833.488}
SPL {X  -156.153, Y  +706.328, Z    +0.000, E1  +392.414, E3 -73837.181}
SPL {X  -159.178, Y  +687.603, Z    +0.000, E1  +378.267, E3 -73839.158}
SPL {X  -159.974, Y  +673.783, Z    +0.000, E1  +364.843, E3 -73839.780}
SPL {X  -159.990, Y  +669.500, Z    +0.000, E1  +360.000, E3 -73839.828}
SPL {X  -159.990, Y  +667.470, Z    +0.000, E1  +355.588, E3 -73839.846}
SPL {X  -159.990, Y  +662.995, Z    +0.000, E1  +343.976, E3 -73839.962}
SPL {X  -159.990, Y  +658.179, Z    +0.000, E1  +331.312, E3 -73840.199}
SPL {X  -159.990, Y  +652.822, Z    +0.000, E1  +319.345, E3 -73840.614}
SPL {X  -159.990, Y  +646.185, Z    +0.000, E1  +308.728, E3 -73841.352}
SPL {X  -159.990, Y  +636.375, Z    +0.000, E1  +299.286, E3 -73842.792}
SPL {X  -159.990, Y  +617.374, Z    +0.000, E1  +291.478, E3 -73847.118}
SPL {X  -159.990, Y  +579.000, Z    +0.000, E1  +286.931, E3 -73858.577}
SPL {X  -157.725, Y  +355.675, Z    +0.000, E1  +284.959, E3 -73955.536}
SPL {X  -142.593, Y  +309.947, Z    +0.000, E1  +282.426, E3 -73949.199}
SPL {X  -142.198, Y  +309.176, Z    +0.000, E1  +283.218, E3 -73958.008}
ENDSPLINE

SPLINE
SPL {X  -142.352, Y  +309.474, Z    +0.000, E1  +284.206, E3 -73967.701}
ENDSPLINE

SPLINE
SPL {X  -141.929, Y  +308.657, Z    +0.000, E1  +285.131, E3 -73976.786}
SPL {X  -140.635, Y  +306.221, Z    +0.000, E1  +286.163, E3 -73987.199}
SPL {X  -138.743, Y  +302.832, Z    +0.000, E1  +287.062, E3 -73996.208}
SPL {X  -135.531, Y  +297.482, Z    +0.000, E1  +287.444, E3 -74002.043}
SPL {X  -132.271, Y  +292.493, Z    +0.000, E1  +287.844, E3 -74007.561}
SPL {X  -128.837, Y  +287.643, Z    +0.000, E1  +288.283, E3 -74012.999}
SPL {X  -125.941, Y  +283.830, Z    +0.000, E1  +288.683, E3 -74017.299}
SPL {X  -124.080, Y  +281.501, Z    +0.000, E1  +288.943, E3 -74019.909}
SPL {X  -120.791, Y  +277.589, Z    +0.000, E1  +289.397, E3 -74024.234}
SPL {X   -74.058, Y  +240.683, Z    +0.000, E1  +305.011, E3 -74181.297}
ENDSPLINE

SPLINE
SPL {X  -130.401, Y  +289.805, Z    +0.000, E1  +307.505, E3 -74338.267}
SPL {X  -152.244, Y  +333.323, Z    +0.000, E1  +320.871, E3 -74355.079}
SPL {X  -158.218, Y  +358.753, Z    +0.000, E1  +336.397, E3 -74359.251}
SPL {X  -159.681, Y  +372.564, Z    +0.000, E1  +347.981, E3 -74360.303}
SPL {X  -159.987, Y  +381.561, Z    +0.000, E1  +356.806, E3 -74360.599}
SPL {X  -159.990, Y  +384.668, Z    +0.000, E1  +360.183, E3 -74360.625}
SPL {X  -159.990, Y  +387.837, Z    +0.000, E1  +367.342, E3 -74360.666}
SPL {X  -159.990, Y  +393.084, Z    +0.000, E1  +380.137, E3 -74360.876}
SPL {X  -159.990, Y  +401.914, Z    +0.000, E1  +400.147, E3 -74361.569}
SPL {X  -159.990, Y  +414.609, Z    +0.000, E1  +416.791, E3 -74363.306}
SPL {X  -159.990, Y  +464.476, Z    +0.000, E1  +431.765, E3 -74376.107}
SPL {X  -158.553, Y  +692.895, Z    +0.000, E1  +434.809, E3 -74474.870}
SPL {X  -156.740, Y  +703.585, Z    +0.000, E1  +434.640, E3 -74482.875}
SPL {X  -154.470, Y  +713.164, Z    +0.000, E1  +434.425, E3 -74490.710}
SPL {X  -151.032, Y  +724.285, Z    +0.000, E1  +434.102, E3 -74500.514}
SPL {X  -147.134, Y  +734.337, Z    +0.000, E1  +433.686, E3 -74510.152}
SPL {X  -143.804, Y  +741.622, Z    +0.000, E1  +433.324, E3 -74517.540}
SPL {X  -140.603, Y  +747.839, Z    +0.000, E1  +432.964, E3 -74524.055}
SPL {X  -137.184, Y  +753.824, Z    +0.000, E1  +432.574, E3 -74530.492}
SPL {X  -133.762, Y  +759.276, Z    +0.000, E1  +432.150, E3 -74536.546}
SPL {X  -130.927, Y  +763.451, Z    +0.000, E1  +431.785, E3 -74541.240}
SPL {X  -126.852, Y  +768.996, Z    +0.000, E1  +431.276, E3 -74547.471}
SPL {X  -122.512, Y  +774.396, Z    +0.000, E1  +430.640, E3 -74553.580}
SPL {X  -119.782, Y  +777.562, Z    +0.000, E1  +430.221, E3 -74557.088}
SPL {X   -71.924, Y  +814.412, Z    +0.000, E1  +415.124, E3 -74713.958}
ENDSPLINE

SPLINE
SPL {X  -132.255, Y  +761.530, Z    +0.000, E1  +413.203, E3 -74877.127}
SPL {X  -150.415, Y  +726.018, Z    +0.000, E1  +402.769, E3 -74890.631}
SPL {X  -156.153, Y  +706.328, Z    +0.000, E1  +392.414, E3 -74894.323}
SPL {X  -159.178, Y  +687.603, Z    +0.000, E1  +378.267, E3 -74896.301}
SPL {X  -159.974, Y  +673.783, Z    +0.000, E1  +364.843, E3 -74896.923}
SPL {X  -159.990, Y  +669.500, Z    +0.000, E1  +360.000, E3 -74896.971}
SPL {X  -159.990, Y  +667.470, Z    +0.000, E1  +355.588, E3 -74896.989}
SPL {X  -159.990, Y  +662.995, Z    +0.000, E1  +343.976, E3 -74897.105}
SPL {X  -159.990, Y  +658.179, Z    +0.000, E1  +331.312, E3 -74897.342}
SPL {X  -159.990, Y  +652.822, Z    +0.000, E1  +319.345, E3 -74897.757}
SPL {X  -159.990, Y  +646.185, Z    +0.000, E1  +308.728, E3 -74898.495}
SPL {X  -159.990, Y  +636.375, Z    +0.000, E1  +299.286, E3 -74899.935}
SPL {X  -159.990, Y  +617.374, Z    +0.000, E1  +291.478, E3 -74904.261}
SPL {X  -159.990, Y  +579.000, Z    +0.000, E1  +286.931, E3 -74915.720}
SPL {X  -157.725, Y  +355.675, Z    +0.000, E1  +284.959, E3 -75012.678}
SPL {X  -142.593, Y  +309.947, Z    +0.000, E1  +282.426, E3 -75006.342}
SPL {X  -142.198, Y  +309.176, Z    +0.000, E1  +283.218, E3 -75015.150}
ENDSPLINE

SPLINE
SPL {X  -142.352, Y  +309.474, Z    +0.000, E1  +284.206, E3 -75024.844}
ENDSPLINE

SPLINE
SPL {X  -141.929, Y  +308.657, Z    +0.000, E1  +285.131, E3 -75033.929}
SPL {X  -140.635, Y  +306.221, Z    +0.000, E1  +286.163, E3 -75044.342}
SPL {X  -138.743, Y  +302.832, Z    +0.000, E1  +287.062, E3 -75053.351}
SPL {X  -135.531, Y  +297.482, Z    +0.000, E1  +287.444, E3 -75059.186}
SPL {X  -132.271, Y  +292.493, Z    +0.000, E1  +287.844, E3 -75064.704}
SPL {X  -128.837, Y  +287.643, Z    +0.000, E1  +288.283, E3 -75070.142}
SPL {X  -125.941, Y  +283.830, Z    +0.000, E1  +288.683, E3 -75074.442}
SPL {X  -124.080, Y  +281.501, Z    +0.000, E1  +288.943, E3 -75077.052}
SPL {X  -120.791, Y  +277.589, Z    +0.000, E1  +289.397, E3 -75081.376}
SPL {X   -74.058, Y  +240.683, Z    +0.000, E1  +305.011, E3 -75238.439}
ENDSPLINE

SPLINE
SPL {X  -130.401, Y  +289.805, Z    +0.000, E1  +307.505, E3 -75395.410}
SPL {X  -152.244, Y  +333.323, Z    +0.000, E1  +320.871, E3 -75412.222}
SPL {X  -158.218, Y  +358.753, Z    +0.000, E1  +336.397, E3 -75416.394}
SPL {X  -159.681, Y  +372.564, Z    +0.000, E1  +347.981, E3 -75417.446}
SPL {X  -159.987, Y  +381.561, Z    +0.000, E1  +356.806, E3 -75417.742}
SPL {X  -159.990, Y  +384.668, Z    +0.000, E1  +360.183, E3 -75417.768}
SPL {X  -159.990, Y  +387.837, Z    +0.000, E1  +367.342, E3 -75417.809}
SPL {X  -159.990, Y  +393.084, Z    +0.000, E1  +380.137, E3 -75418.018}
SPL {X  -159.990, Y  +401.914, Z    +0.000, E1  +400.147, E3 -75418.712}
SPL {X  -159.990, Y  +414.609, Z    +0.000, E1  +416.791, E3 -75420.449}
SPL {X  -159.990, Y  +464.476, Z    +0.000, E1  +431.765, E3 -75433.250}
SPL {X  -158.553, Y  +692.895, Z    +0.000, E1  +434.809, E3 -75532.013}
SPL {X  -156.740, Y  +703.585, Z    +0.000, E1  +434.640, E3 -75540.018}
SPL {X  -154.470, Y  +713.164, Z    +0.000, E1  +434.425, E3 -75547.853}
SPL {X  -151.032, Y  +724.285, Z    +0.000, E1  +434.102, E3 -75557.657}
SPL {X  -147.134, Y  +734.337, Z    +0.000, E1  +433.686, E3 -75567.295}
SPL {X  -143.804, Y  +741.622, Z    +0.000, E1  +433.324, E3 -75574.682}
SPL {X  -140.603, Y  +747.839, Z    +0.000, E1  +432.964, E3 -75581.198}
SPL {X  -137.184, Y  +753.824, Z    +0.000, E1  +432.574, E3 -75587.635}
SPL {X  -133.762, Y  +759.276, Z    +0.000, E1  +432.150, E3 -75593.688}
SPL {X  -130.927, Y  +763.451, Z    +0.000, E1  +431.785, E3 -75598.383}
SPL {X  -126.852, Y  +768.996, Z    +0.000, E1  +431.276, E3 -75604.614}
SPL {X  -122.512, Y  +774.396, Z    +0.000, E1  +430.640, E3 -75610.723}
SPL {X  -119.782, Y  +777.562, Z    +0.000, E1  +430.221, E3 -75614.230}
SPL {X   -71.924, Y  +814.412, Z    +0.000, E1  +415.124, E3 -75771.100}
ENDSPLINE

SPLINE
SPL {X  -132.255, Y  +761.530, Z    +0.000, E1  +413.203, E3 -75934.270}
SPL {X  -150.415, Y  +726.018, Z    +0.000, E1  +402.769, E3 -75947.774}
SPL {X  -156.153, Y  +706.328, Z    +0.000, E1  +392.414, E3 -75951.466}
SPL {X  -159.178, Y  +687.603, Z    +0.000, E1  +378.267, E3 -75953.444}
SPL {X  -159.974, Y  +673.783, Z    +0.000, E1  +364.843, E3 -75954.066}
SPL {X  -159.990, Y  +669.500, Z    +0.000, E1  +360.000, E3 -75954.114}
SPL {X  -159.990, Y  +667.470, Z    +0.000, E1  +355.588, E3 -75954.132}
SPL {X  -159.990, Y  +662.995, Z    +0.000, E1  +343.976, E3 -75954.248}
SPL {X  -159.990, Y  +658.179, Z    +0.000, E1  +331.312, E3 -75954.485}
SPL {X  -159.990, Y  +652.822, Z    +0.000, E1  +319.345, E3 -75954.899}
SPL {X  -159.990, Y  +646.185, Z    +0.000, E1  +308.728, E3 -75955.638}
SPL {X  -159.990, Y  +632.371, Z    +0.000, E1  +297.040, E3 -75957.991}
SPL {X  -159.990, Y  +579.000, Z    +0.000, E1  +286.931, E3 -75972.863}
SPL {X  -157.725, Y  +355.675, Z    +0.000, E1  +284.959, E3 -76069.821}
SPL {X  -142.593, Y  +309.947, Z    +0.000, E1  +282.426, E3 -76063.485}
SPL {X  -142.198, Y  +309.176, Z    +0.000, E1  +283.218, E3 -76072.293}
ENDSPLINE

SPLINE
SPL {X  -142.352, Y  +309.474, Z    +0.000, E1  +284.206, E3 -76081.987}
ENDSPLINE

SPLINE
SPL {X  -141.553, Y  +307.937, Z    +0.000, E1  +285.290, E3 -76093.003}
SPL {X  -140.562, Y  +306.086, Z    +0.000, E1  +286.440, E3 -76103.697}
SPL {X  -138.743, Y  +302.832, Z    +0.000, E1  +287.062, E3 -76110.494}
SPL {X  -135.531, Y  +297.482, Z    +0.000, E1  +287.444, E3 -76116.329}
SPL {X  -132.271, Y  +292.493, Z    +0.000, E1  +287.844, E3 -76121.847}
SPL {X  -128.837, Y  +287.643, Z    +0.000, E1  +288.283, E3 -76127.285}
SPL {X  -124.965, Y  +282.598, Z    +0.000, E1  +288.800, E3 -76132.946}
SPL {X  -120.791, Y  +277.589, Z    +0.000, E1  +289.397, E3 -76138.519}
SPL {X   -74.058, Y  +240.683, Z    +0.000, E1  +305.011, E3 -76295.582}
ENDSPLINE

SPLINE
SPL {X  -130.401, Y  +289.805, Z    +0.000, E1  +307.505, E3 -76452.553}
SPL {X  -148.502, Y  +322.968, Z    +0.000, E1  +316.497, E3 -76466.873}
SPL {X  -154.800, Y  +342.080, Z    +0.000, E1  +325.471, E3 -76471.177}
SPL {X  -158.218, Y  +358.753, Z    +0.000, E1  +336.397, E3 -76473.537}
SPL {X  -159.681, Y  +372.564, Z    +0.000, E1  +347.981, E3 -76474.589}
SPL {X  -159.987, Y  +381.561, Z    +0.000, E1  +356.806, E3 -76474.885}
SPL {X  -159.990, Y  +384.668, Z    +0.000, E1  +360.183, E3 -76474.911}
SPL {X  -159.990, Y  +387.837, Z    +0.000, E1  +367.342, E3 -76474.951}
SPL {X  -159.990, Y  +393.084, Z    +0.000, E1  +380.137, E3 -76475.161}
SPL {X  -159.990, Y  +401.914, Z    +0.000, E1  +400.147, E3 -76475.855}
SPL {X  -159.990, Y  +414.609, Z    +0.000, E1  +416.791, E3 -76477.592}
SPL {X  -159.990, Y  +464.476, Z    +0.000, E1  +431.765, E3 -76490.393}
SPL {X  -157.643, Y  +698.802, Z    +0.000, E1  +434.751, E3 -76593.407}
SPL {X  -154.470, Y  +713.164, Z    +0.000, E1  +434.425, E3 -76604.996}
SPL {X  -151.032, Y  +724.285, Z    +0.000, E1  +434.102, E3 -76614.800}
SPL {X  -147.134, Y  +734.337, Z    +0.000, E1  +433.686, E3 -76624.437}
SPL {X  -143.804, Y  +741.622, Z    +0.000, E1  +433.324, E3 -76631.825}
SPL {X  -140.603, Y  +747.839, Z    +0.000, E1  +432.964, E3 -76638.341}
SPL {X  -137.184, Y  +753.824, Z    +0.000, E1  +432.574, E3 -76644.778}
SPL {X  -133.762, Y  +759.276, Z    +0.000, E1  +432.150, E3 -76650.831}
SPL {X  -130.927, Y  +763.451, Z    +0.000, E1  +431.785, E3 -76655.526}
SPL {X  -128.105, Y  +767.343, Z    +0.000, E1  +431.419, E3 -76659.915}
SPL {X  -124.554, Y  +771.914, Z    +0.000, E1  +430.935, E3 -76665.086}
SPL {X  -120.687, Y  +776.531, Z    +0.000, E1  +430.379, E3 -76670.219}
SPL {X   -71.924, Y  +814.412, Z    +0.000, E1  +415.124, E3 -76828.243}
ENDSPLINE

SPLINE
SPL {X  -132.255, Y  +761.530, Z    +0.000, E1  +413.203, E3 -76991.413}
SPL {X  -150.415, Y  +726.018, Z    +0.000, E1  +402.769, E3 -77004.917}
SPL {X  -156.153, Y  +706.328, Z    +0.000, E1  +392.414, E3 -77008.609}
SPL {X  -159.178, Y  +687.603, Z    +0.000, E1  +378.267, E3 -77010.587}
SPL {X  -159.974, Y  +673.783, Z    +0.000, E1  +364.843, E3 -77011.209}
SPL {X  -159.990, Y  +669.500, Z    +0.000, E1  +360.000, E3 -77011.256}
SPL {X  -159.990, Y  +667.470, Z    +0.000, E1  +355.588, E3 -77011.274}
SPL {X  -159.990, Y  +662.995, Z    +0.000, E1  +343.976, E3 -77011.391}
SPL {X  -159.990, Y  +658.179, Z    +0.000, E1  +331.312, E3 -77011.628}
SPL {X  -159.990, Y  +652.822, Z    +0.000, E1  +319.345, E3 -77012.042}
SPL {X  -159.990, Y  +646.185, Z    +0.000, E1  +308.728, E3 -77012.781}
SPL {X  -159.990, Y  +632.371, Z    +0.000, E1  +297.040, E3 -77015.134}
SPL {X  -159.990, Y  +579.000, Z    +0.000, E1  +286.931, E3 -77030.006}
SPL {X  -157.725, Y  +355.675, Z    +0.000, E1  +284.959, E3 -77126.964}
SPL {X  -142.593, Y  +309.947, Z    +0.000, E1  +282.426, E3 -77120.628}
SPL {X  -142.198, Y  +309.176, Z    +0.000, E1  +283.218, E3 -77129.436}
ENDSPLINE

SPLINE
SPL {X  -142.352, Y  +309.474, Z    +0.000, E1  +284.206, E3 -77139.130}
ENDSPLINE

SPLINE
SPL {X  -141.553, Y  +307.937, Z    +0.000, E1  +285.290, E3 -77150.146}
SPL {X  -140.562, Y  +306.086, Z    +0.000, E1  +286.440, E3 -77160.839}
SPL {X  -138.743, Y  +302.832, Z    +0.000, E1  +287.062, E3 -77167.637}
SPL {X  -135.531, Y  +297.482, Z    +0.000, E1  +287.444, E3 -77173.471}
SPL {X  -132.271, Y  +292.493, Z    +0.000, E1  +287.844, E3 -77178.990}
SPL {X  -128.837, Y  +287.643, Z    +0.000, E1  +288.283, E3 -77184.428}
SPL {X  -124.965, Y  +282.598, Z    +0.000, E1  +288.800, E3 -77190.089}
SPL {X  -120.791, Y  +277.589, Z    +0.000, E1  +289.397, E3 -77195.662}
SPL {X   -74.058, Y  +240.683, Z    +0.000, E1  +305.011, E3 -77352.725}
ENDSPLINE

SPLINE
SPL {X  -130.401, Y  +289.805, Z    +0.000, E1  +307.505, E3 -77509.696}
SPL {X  -148.502, Y  +322.968, Z    +0.000, E1  +316.497, E3 -77524.016}
SPL {X  -154.800, Y  +342.080, Z    +0.000, E1  +325.471, E3 -77528.320}
SPL {X  -158.218, Y  +358.753, Z    +0.000, E1  +336.397, E3 -77530.680}
SPL {X  -159.681, Y  +372.564, Z    +0.000, E1  +347.981, E3 -77531.731}
SPL {X  -159.987, Y  +381.561, Z    +0.000, E1  +356.806, E3 -77532.028}
SPL {X  -159.990, Y  +384.668, Z    +0.000, E1  +360.183, E3 -77532.054}
SPL {X  -159.990, Y  +387.837, Z    +0.000, E1  +367.342, E3 -77532.094}
SPL {X  -159.990, Y  +393.084, Z    +0.000, E1  +380.137, E3 -77532.304}
SPL {X  -159.990, Y  +401.914, Z    +0.000, E1  +400.147, E3 -77532.998}
SPL {X  -159.990, Y  +414.609, Z    +0.000, E1  +416.791, E3 -77534.735}
SPL {X  -159.990, Y  +464.476, Z    +0.000, E1  +431.765, E3 -77547.536}
SPL {X  -157.643, Y  +698.802, Z    +0.000, E1  +434.751, E3 -77650.550}
SPL {X  -154.470, Y  +713.164, Z    +0.000, E1  +434.425, E3 -77662.139}
SPL {X  -151.032, Y  +724.285, Z    +0.000, E1  +434.102, E3 -77671.943}
SPL {X  -147.134, Y  +734.337, Z    +0.000, E1  +433.686, E3 -77681.580}
SPL {X  -143.804, Y  +741.622, Z    +0.000, E1  +433.324, E3 -77688.968}
SPL {X  -140.603, Y  +747.839, Z    +0.000, E1  +432.964, E3 -77695.484}
SPL {X  -137.184, Y  +753.824, Z    +0.000, E1  +432.574, E3 -77701.920}
SPL {X  -133.762, Y  +759.276, Z    +0.000, E1  +432.150, E3 -77707.974}
SPL {X  -130.927, Y  +763.451, Z    +0.000, E1  +431.785, E3 -77712.669}
SPL {X  -126.852, Y  +768.996, Z    +0.000, E1  +431.276, E3 -77718.900}
SPL {X  -122.512, Y  +774.396, Z    +0.000, E1  +430.640, E3 -77725.009}
SPL {X  -119.782, Y  +777.562, Z    +0.000, E1  +430.221, E3 -77728.516}
SPL {X   -71.924, Y  +814.412, Z    +0.000, E1  +415.124, E3 -77885.386}
ENDSPLINE

SPLINE
SPL {X  -132.255, Y  +761.530, Z    +0.000, E1  +413.203, E3 -78048.556}
SPL {X  -150.415, Y  +726.018, Z    +0.000, E1  +402.769, E3 -78062.060}
SPL {X  -156.153, Y  +706.328, Z    +0.000, E1  +392.414, E3 -78065.752}
SPL {X  -159.178, Y  +687.603, Z    +0.000, E1  +378.267, E3 -78067.730}
SPL {X  -159.974, Y  +673.783, Z    +0.000, E1  +364.843, E3 -78068.352}
SPL {X  -159.990, Y  +669.500, Z    +0.000, E1  +360.000, E3 -78068.399}
SPL {X  -159.990, Y  +667.470, Z    +0.000, E1  +355.588, E3 -78068.417}
SPL {X  -159.990, Y  +662.995, Z    +0.000, E1  +343.976, E3 -78068.534}
SPL {X  -159.990, Y  +658.179, Z    +0.000, E1  +331.312, E3 -78068.770}
SPL {X  -159.990, Y  +652.822, Z    +0.000, E1  +319.345, E3 -78069.185}
SPL {X  -159.990, Y  +646.185, Z    +0.000, E1  +308.728, E3 -78069.924}
SPL {X  -159.990, Y  +636.375, Z    +0.000, E1  +299.286, E3 -78071.363}
SPL {X  -159.990, Y  +617.374, Z    +0.000, E1  +291.478, E3 -78075.690}
SPL {X  -159.990, Y  +579.000, Z    +0.000, E1  +286.931, E3 -78087.149}
SPL {X  -157.725, Y  +355.675, Z    +0.000, E1  +284.959, E3 -78184.107}
SPL {X  -142.593, Y  +309.947, Z    +0.000, E1  +282.426, E3 -78177.770}
SPL {X  -142.198, Y  +309.176, Z    +0.000, E1  +283.218, E3 -78186.579}
ENDSPLINE

SPLINE
SPL {X  -142.352, Y  +309.474, Z    +0.000, E1  +284.206, E3 -78196.273}
ENDSPLINE

SPLINE
SPL {X  -141.929, Y  +308.657, Z    +0.000, E1  +285.131, E3 -78205.358}
SPL {X  -140.635, Y  +306.221, Z    +0.000, E1  +286.163, E3 -78215.770}
SPL {X  -138.743, Y  +302.832, Z    +0.000, E1  +287.062, E3 -78224.780}
SPL {X  -135.531, Y  +297.482, Z    +0.000, E1  +287.444, E3 -78230.614}
SPL {X  -132.271, Y  +292.493, Z    +0.000, E1  +287.844, E3 -78236.133}
SPL {X  -128.837, Y  +287.643, Z    +0.000, E1  +288.283, E3 -78241.570}
SPL {X  -125.941, Y  +283.830, Z    +0.000, E1  +288.683, E3 -78245.870}
SPL {X  -124.080, Y  +281.501, Z    +0.000, E1  +288.943, E3 -78248.481}
SPL {X  -120.791, Y  +277.589, Z    +0.000, E1  +289.397, E3 -78252.805}
SPL {X   -74.058, Y  +240.683, Z    +0.000, E1  +305.011, E3 -78409.868}
ENDSPLINE

SPLINE
SPL {X  -130.401, Y  +289.805, Z    +0.000, E1  +307.505, E3 -78566.839}
SPL {X  -152.244, Y  +333.323, Z    +0.000, E1  +320.871, E3 -78583.650}
SPL {X  -158.218, Y  +358.753, Z    +0.000, E1  +336.397, E3 -78587.823}
SPL {X  -159.681, Y  +372.564, Z    +0.000, E1  +347.981, E3 -78588.874}
SPL {X  -159.987, Y  +381.561, Z    +0.000, E1  +356.806, E3 -78589.171}
SPL {X  -159.990, Y  +384.668, Z    +0.000, E1  +360.183, E3 -78589.196}
SPL {X  -159.990, Y  +387.837, Z    +0.000, E1  +367.342, E3 -78589.237}
SPL {X  -159.990, Y  +393.084, Z    +0.000, E1  +380.137, E3 -78589.447}
SPL {X  -159.990, Y  +401.914, Z    +0.000, E1  +400.147, E3 -78590.141}
SPL {X  -159.990, Y  +414.609, Z    +0.000, E1  +416.791, E3 -78591.877}
SPL {X  -159.990, Y  +464.476, Z    +0.000, E1  +431.765, E3 -78604.678}
SPL {X  -158.553, Y  +692.895, Z    +0.000, E1  +434.809, E3 -78703.442}
SPL {X  -156.740, Y  +703.585, Z    +0.000, E1  +434.640, E3 -78711.447}
SPL {X  -154.470, Y  +713.164, Z    +0.000, E1  +434.425, E3 -78719.282}
SPL {X  -151.032, Y  +724.285, Z    +0.000, E1  +434.102, E3 -78729.086}
SPL {X  -147.134, Y  +734.337, Z    +0.000, E1  +433.686, E3 -78738.723}
SPL {X  -143.804, Y  +741.622, Z    +0.000, E1  +433.324, E3 -78746.111}
SPL {X  -140.603, Y  +747.839, Z    +0.000, E1  +432.964, E3 -78752.627}
SPL {X  -137.184, Y  +753.824, Z    +0.000, E1  +432.574, E3 -78759.063}
SPL {X  -133.762, Y  +759.276, Z    +0.000, E1  +432.150, E3 -78765.117}
SPL {X  -130.927, Y  +763.451, Z    +0.000, E1  +431.785, E3 -78769.812}
SPL {X  -126.852, Y  +768.996, Z    +0.000, E1  +431.276, E3 -78776.042}
SPL {X  -122.512, Y  +774.396, Z    +0.000, E1  +430.640, E3 -78782.152}
SPL {X  -119.782, Y  +777.562, Z    +0.000, E1  +430.221, E3 -78785.659}
SPL {X   -71.924, Y  +814.412, Z    +0.000, E1  +415.124, E3 -78942.529}
ENDSPLINE

SPLINE
SPL {X  -132.255, Y  +761.530, Z    +0.000, E1  +413.203, E3 -79105.699}
SPL {X  -150.415, Y  +726.018, Z    +0.000, E1  +402.769, E3 -79119.203}
SPL {X  -156.153, Y  +706.328, Z    +0.000, E1  +392.414, E3 -79122.895}
SPL {X  -159.178, Y  +687.603, Z    +0.000, E1  +378.267, E3 -79124.873}
SPL {X  -159.974, Y  +673.783, Z    +0.000, E1  +364.843, E3 -79125.495}
SPL {X  -159.990, Y  +669.500, Z    +0.000, E1  +360.000, E3 -79125.542}
SPL {X  -159.990, Y  +667.470, Z    +0.000, E1  +355.588, E3 -79125.560}
SPL {X  -159.990, Y  +662.995, Z    +0.000, E1  +343.976, E3 -79125.677}
SPL {X  -159.990, Y  +658.179, Z    +0.000, E1  +331.312, E3 -79125.913}
SPL {X  -159.990, Y  +652.822, Z    +0.000, E1  +319.345, E3 -79126.328}
SPL {X  -159.990, Y  +646.185, Z    +0.000, E1  +308.728, E3 -79127.067}
SPL {X  -159.990, Y  +636.375, Z    +0.000, E1  +299.286, E3 -79128.506}
SPL {X  -159.990, Y  +617.374, Z    +0.000, E1  +291.478, E3 -79132.833}
SPL {X  -159.990, Y  +579.000, Z    +0.000, E1  +286.931, E3 -79144.292}
SPL {X  -157.725, Y  +355.675, Z    +0.000, E1  +284.959, E3 -79241.250}
SPL {X  -142.593, Y  +309.947, Z    +0.000, E1  +282.426, E3 -79234.913}
SPL {X  -142.198, Y  +309.176, Z    +0.000, E1  +283.218, E3 -79243.722}
ENDSPLINE

SPLINE
SPL {X  -142.352, Y  +309.474, Z    +0.000, E1  +284.206, E3 -79253.415}
ENDSPLINE

SPLINE
SPL {X  -141.553, Y  +307.937, Z    +0.000, E1  +285.290, E3 -79264.431}
SPL {X  -140.562, Y  +306.086, Z    +0.000, E1  +286.440, E3 -79275.125}
SPL {X  -138.743, Y  +302.832, Z    +0.000, E1  +287.062, E3 -79281.923}
SPL {X  -135.531, Y  +297.482, Z    +0.000, E1  +287.444, E3 -79287.757}
SPL {X  -132.271, Y  +292.493, Z    +0.000, E1  +287.844, E3 -79293.276}
SPL {X  -128.837, Y  +287.643, Z    +0.000, E1  +288.283, E3 -79298.713}
SPL {X  -125.941, Y  +283.830, Z    +0.000, E1  +288.683, E3 -79303.013}
SPL {X  -124.080, Y  +281.501, Z    +0.000, E1  +288.943, E3 -79305.624}
SPL {X  -120.791, Y  +277.589, Z    +0.000, E1  +289.397, E3 -79309.948}
SPL {X   -74.058, Y  +240.683, Z    +0.000, E1  +305.011, E3 -79467.011}
ENDSPLINE

SPLINE
SPL {X  -130.401, Y  +289.805, Z    +0.000, E1  +307.505, E3 -79623.982}
SPL {X  -148.502, Y  +322.968, Z    +0.000, E1  +316.497, E3 -79638.302}
SPL {X  -154.800, Y  +342.080, Z    +0.000, E1  +325.471, E3 -79642.606}
SPL {X  -158.218, Y  +358.753, Z    +0.000, E1  +336.397, E3 -79644.966}
SPL {X  -159.681, Y  +372.564, Z    +0.000, E1  +347.981, E3 -79646.017}
SPL {X  -159.987, Y  +381.561, Z    +0.000, E1  +356.806, E3 -79646.314}
SPL {X  -159.990, Y  +384.668, Z    +0.000, E1  +360.183, E3 -79646.339}
SPL {X  -159.990, Y  +387.837, Z    +0.000, E1  +367.342, E3 -79646.380}
SPL {X  -159.990, Y  +393.084, Z    +0.000, E1  +380.137, E3 -79646.590}
SPL {X  -159.990, Y  +401.914, Z    +0.000, E1  +400.147, E3 -79647.283}
SPL {X  -159.990, Y  +414.609, Z    +0.000, E1  +416.791, E3 -79649.020}
SPL {X  -159.990, Y  +464.476, Z    +0.000, E1  +431.765, E3 -79661.821}
SPL {X  -157.643, Y  +698.802, Z    +0.000, E1  +434.751, E3 -79764.836}
SPL {X  -154.470, Y  +713.164, Z    +0.000, E1  +434.425, E3 -79776.425}
SPL {X  -152.098, Y  +721.129, Z    +0.000, E1  +434.190, E3 -79783.397}
SPL {X  -148.128, Y  +731.956, Z    +0.000, E1  +433.814, E3 -79793.478}
SPL {X  -143.804, Y  +741.622, Z    +0.000, E1  +433.324, E3 -79803.254}
SPL {X  -140.603, Y  +747.839, Z    +0.000, E1  +432.964, E3 -79809.769}
SPL {X  -137.184, Y  +753.824, Z    +0.000, E1  +432.574, E3 -79816.206}
SPL {X  -133.762, Y  +759.276, Z    +0.000, E1  +432.150, E3 -79822.260}
SPL {X  -130.927, Y  +763.451, Z    +0.000, E1  +431.785, E3 -79826.954}
SPL {X  -128.105, Y  +767.343, Z    +0.000, E1  +431.419, E3 -79831.343}
SPL {X  -124.554, Y  +771.914, Z    +0.000, E1  +430.935, E3 -79836.514}
SPL {X  -120.687, Y  +776.531, Z    +0.000, E1  +430.379, E3 -79841.647}
SPL {X   -71.924, Y  +814.412, Z    +0.000, E1  +415.124, E3 -79999.672}
ENDSPLINE

SPLINE
SPL {X  -132.255, Y  +761.530, Z    +0.000, E1  +413.203, E3 -80162.842}
SPL {X  -150.415, Y  +726.018, Z    +0.000, E1  +402.769, E3 -80176.346}
SPL {X  -157.206, Y  +701.216, Z    +0.000, E1  +389.056, E3 -80180.684}
SPL {X  -159.772, Y  +679.843, Z    +0.000, E1  +371.089, E3 -80182.448}
SPL {X  -159.990, Y  +669.381, Z    +0.000, E1  +359.965, E3 -80182.685}
SPL {X  -159.990, Y  +666.412, Z    +0.000, E1  +352.765, E3 -80182.717}
SPL {X  -159.990, Y  +662.995, Z    +0.000, E1  +343.976, E3 -80182.819}
SPL {X  -159.990, Y  +658.179, Z    +0.000, E1  +331.312, E3 -80183.056}
SPL {X  -159.990, Y  +652.822, Z    +0.000, E1  +319.345, E3 -80183.471}
SPL {X  -159.990, Y  +646.185, Z    +0.000, E1  +308.728, E3 -80184.210}
SPL {X  -159.990, Y  +632.371, Z    +0.000, E1  +297.040, E3 -80186.562}
SPL {X  -159.990, Y  +579.000, Z    +0.000, E1  +286.931, E3 -80201.434}
SPL {X  -157.725, Y  +355.675, Z    +0.000, E1  +284.959, E3 -80298.393}
SPL {X  -142.593, Y  +309.947, Z    +0.000, E1  +282.426, E3 -80292.056}
SPL {X  -142.198, Y  +309.176, Z    +0.000, E1  +283.218, E3 -80300.865}
ENDSPLINE

SPLINE
SPL {X  -142.352, Y  +309.474, Z    +0.000, E1  +284.206, E3 -80310.558}
ENDSPLINE

SPLINE
SPL {X  -141.929, Y  +308.657, Z    +0.000, E1  +285.131, E3 -80319.644}
SPL {X  -140.635, Y  +306.221, Z    +0.000, E1  +286.163, E3 -80330.056}
SPL {X  -138.743, Y  +302.832, Z    +0.000, E1  +287.062, E3 -80339.065}
SPL {X  -135.531, Y  +297.482, Z    +0.000, E1  +287.444, E3 -80344.900}
SPL {X  -132.271, Y  +292.493, Z    +0.000, E1  +287.844, E3 -80350.418}
SPL {X  -128.837, Y  +287.643, Z    +0.000, E1  +288.283, E3 -80355.856}
SPL {X  -124.965, Y  +282.598, Z    +0.000, E1  +288.800, E3 -80361.518}
SPL {X  -120.791, Y  +277.589, Z    +0.000, E1  +289.397, E3 -80367.091}
SPL {X   -74.058, Y  +240.683, Z    +0.000, E1  +305.011, E3 -80524.154}
ENDSPLINE

SPLINE
SPL {X  -130.401, Y  +289.805, Z    +0.000, E1  +307.505, E3 -80681.125}
SPL {X  -148.502, Y  +322.968, Z    +0.000, E1  +316.497, E3 -80695.445}
SPL {X  -154.800, Y  +342.080, Z    +0.000, E1  +325.471, E3 -80699.749}
SPL {X  -158.218, Y  +358.753, Z    +0.000, E1  +336.397, E3 -80702.108}
SPL {X  -159.681, Y  +372.564, Z    +0.000, E1  +347.981, E3 -80703.160}
SPL {X  -159.987, Y  +381.561, Z    +0.000, E1  +356.806, E3 -80703.456}
SPL {X  -159.990, Y  +384.668, Z    +0.000, E1  +360.183, E3 -80703.482}
SPL {X  -159.990, Y  +387.837, Z    +0.000, E1  +367.342, E3 -80703.523}
SPL {X  -159.990, Y  +393.084, Z    +0.000, E1  +380.137, E3 -80703.733}
SPL {X  -159.990, Y  +401.914, Z    +0.000, E1  +400.147, E3 -80704.426}
SPL {X  -159.990, Y  +414.609, Z    +0.000, E1  +416.791, E3 -80706.163}
SPL {X  -159.990, Y  +464.476, Z    +0.000, E1  +431.765, E3 -80718.964}
SPL {X  -157.643, Y  +698.802, Z    +0.000, E1  +434.751, E3 -80821.979}
SPL {X  -154.470, Y  +713.164, Z    +0.000, E1  +434.425, E3 -80833.568}
SPL {X  -151.032, Y  +724.285, Z    +0.000, E1  +434.102, E3 -80843.371}
SPL {X  -147.134, Y  +734.337, Z    +0.000, E1  +433.686, E3 -80853.009}
SPL {X  -143.804, Y  +741.622, Z    +0.000, E1  +433.324, E3 -80860.397}
SPL {X  -140.603, Y  +747.839, Z    +0.000, E1  +432.964, E3 -80866.912}
SPL {X  -137.184, Y  +753.824, Z    +0.000, E1  +432.574, E3 -80873.349}
SPL {X  -133.762, Y  +759.276, Z    +0.000, E1  +432.150, E3 -80879.403}
SPL {X  -130.927, Y  +763.451, Z    +0.000, E1  +431.785, E3 -80884.097}
SPL {X  -128.105, Y  +767.343, Z    +0.000, E1  +431.419, E3 -80888.486}
SPL {X  -124.554, Y  +771.914, Z    +0.000, E1  +430.935, E3 -80893.657}
SPL {X  -120.892, Y  +776.295, Z    +0.000, E1  +430.404, E3 -80898.541}
SPL {X  -118.039, Y  +779.498, Z    +0.000, E1  +429.949, E3 -80902.059}
SPL {X   -71.924, Y  +814.412, Z    +0.000, E1  +415.124, E3 -81056.815}
ENDSPLINE

SPLINE
SPL {X  -132.255, Y  +761.530, Z    +0.000, E1  +413.203, E3 -81219.984}
SPL {X  -150.415, Y  +726.018, Z    +0.000, E1  +402.769, E3 -81233.488}
SPL {X  -156.153, Y  +706.328, Z    +0.000, E1  +392.414, E3 -81237.181}
SPL {X  -159.178, Y  +687.603, Z    +0.000, E1  +378.267, E3 -81239.158}
SPL {X  -159.974, Y  +673.783, Z    +0.000, E1  +364.843, E3 -81239.780}
SPL {X  -159.990, Y  +669.500, Z    +0.000, E1  +360.000, E3 -81239.828}
SPL {X  -159.990, Y  +667.470, Z    +0.000, E1  +355.588, E3 -81239.846}
SPL {X  -159.990, Y  +662.995, Z    +0.000, E1  +343.976, E3 -81239.962}
SPL {X  -159.990, Y  +658.179, Z    +0.000, E1  +331.312, E3 -81240.199}
SPL {X  -159.990, Y  +652.822, Z    +0.000, E1  +319.345, E3 -81240.614}
SPL {X  -159.990, Y  +646.185, Z    +0.000, E1  +308.728, E3 -81241.352}
SPL {X  -159.990, Y  +636.375, Z    +0.000, E1  +299.286, E3 -81242.792}
SPL {X  -159.990, Y  +617.374, Z    +0.000, E1  +291.478, E3 -81247.118}
SPL {X  -159.990, Y  +579.000, Z    +0.000, E1  +286.931, E3 -81258.577}
SPL {X  -157.725, Y  +355.675, Z    +0.000, E1  +284.959, E3 -81355.536}
SPL {X  -142.593, Y  +309.947, Z    +0.000, E1  +282.426, E3 -81349.199}
SPL {X  -142.198, Y  +309.176, Z    +0.000, E1  +283.218, E3 -81358.008}
ENDSPLINE

SPLINE
SPL {X  -142.352, Y  +309.474, Z    +0.000, E1  +284.206, E3 -81367.701}
ENDSPLINE

SPLINE
SPL {X  -141.553, Y  +307.937, Z    +0.000, E1  +285.290, E3 -81378.717}
SPL {X  -140.562, Y  +306.086, Z    +0.000, E1  +286.440, E3 -81389.411}
SPL {X  -138.743, Y  +302.832, Z    +0.000, E1  +287.062, E3 -81396.208}
SPL {X  -135.531, Y  +297.482, Z    +0.000, E1  +287.444, E3 -81402.043}
SPL {X  -132.271, Y  +292.493, Z    +0.000, E1  +287.844, E3 -81407.561}
SPL {X  -128.837, Y  +287.643, Z    +0.000, E1  +288.283, E3 -81412.999}
SPL {X  -125.941, Y  +283.830, Z    +0.000, E1  +288.683, E3 -81417.299}
SPL {X  -124.080, Y  +281.501, Z    +0.000, E1  +288.943, E3 -81419.909}
SPL {X  -120.791, Y  +277.589, Z    +0.000, E1  +289.397, E3 -81424.234}
SPL {X   -74.058, Y  +240.683, Z    +0.000, E1  +305.011, E3 -81581.297}
ENDSPLINE

SPLINE
SPL {X  -130.401, Y  +289.805, Z    +0.000, E1  +307.505, E3 -81738.267}
SPL {X  -152.244, Y  +333.323, Z    +0.000, E1  +320.871, E3 -81755.079}
SPL {X  -158.218, Y  +358.753, Z    +0.000, E1  +336.397, E3 -81759.251}
SPL {X  -159.681, Y  +372.564, Z    +0.000, E1  +347.981, E3 -81760.303}
SPL {X  -159.987, Y  +381.561, Z    +0.000, E1  +356.806, E3 -81760.599}
SPL {X  -159.990, Y  +384.668, Z    +0.000, E1  +360.183, E3 -81760.625}
SPL {X  -159.990, Y  +387.837, Z    +0.000, E1  +367.342, E3 -81760.666}
SPL {X  -159.990, Y  +393.084, Z    +0.000, E1  +380.137, E3 -81760.876}
SPL {X  -159.990, Y  +401.914, Z    +0.000, E1  +400.147, E3 -81761.569}
SPL {X  -159.990, Y  +414.609, Z    +0.000, E1  +416.791, E3 -81763.306}
SPL {X  -159.990, Y  +464.476, Z    +0.000, E1  +431.765, E3 -81776.107}
SPL {X  -157.643, Y  +698.802, Z    +0.000, E1  +434.751, E3 -81879.122}
SPL {X  -154.470, Y  +713.164, Z    +0.000, E1  +434.425, E3 -81890.710}
SPL {X  -151.032, Y  +724.285, Z    +0.000, E1  +434.102, E3 -81900.514}
SPL {X  -147.134, Y  +734.337, Z    +0.000, E1  +433.686, E3 -81910.152}
SPL {X  -143.804, Y  +741.622, Z    +0.000, E1  +433.324, E3 -81917.540}
SPL {X  -140.603, Y  +747.839, Z    +0.000, E1  +432.964, E3 -81924.055}
SPL {X  -137.184, Y  +753.824, Z    +0.000, E1  +432.574, E3 -81930.492}
SPL {X  -133.762, Y  +759.276, Z    +0.000, E1  +432.150, E3 -81936.546}
SPL {X  -130.927, Y  +763.451, Z    +0.000, E1  +431.785, E3 -81941.240}
SPL {X  -128.105, Y  +767.343, Z    +0.000, E1  +431.419, E3 -81945.629}
SPL {X  -124.554, Y  +771.914, Z    +0.000, E1  +430.935, E3 -81950.800}
SPL {X  -120.687, Y  +776.531, Z    +0.000, E1  +430.379, E3 -81955.933}
SPL {X   -71.924, Y  +814.412, Z    +0.000, E1  +415.124, E3 -82113.958}
ENDSPLINE

SPLINE
SPL {X  -132.255, Y  +761.530, Z    +0.000, E1  +413.203, E3 -82277.127}
SPL {X  -150.415, Y  +726.018, Z    +0.000, E1  +402.769, E3 -82290.631}
SPL {X  -156.153, Y  +706.328, Z    +0.000, E1  +392.414, E3 -82294.323}
SPL {X  -159.178, Y  +687.603, Z    +0.000, E1  +378.267, E3 -82296.301}
SPL {X  -159.974, Y  +673.783, Z    +0.000, E1  +364.843, E3 -82296.923}
SPL {X  -159.990, Y  +669.500, Z    +0.000, E1  +360.000, E3 -82296.971}
SPL {X  -159.990, Y  +667.470, Z    +0.000, E1  +355.588, E3 -82296.989}
SPL {X  -159.990, Y  +662.995, Z    +0.000, E1  +343.976, E3 -82297.105}
SPL {X  -159.990, Y  +658.179, Z    +0.000, E1  +331.312, E3 -82297.342}
SPL {X  -159.990, Y  +652.822, Z    +0.000, E1  +319.345, E3 -82297.757}
SPL {X  -159.990, Y  +646.185, Z    +0.000, E1  +308.728, E3 -82298.495}
SPL {X  -159.990, Y  +632.371, Z    +0.000, E1  +297.040, E3 -82300.848}
SPL {X  -159.990, Y  +579.000, Z    +0.000, E1  +286.931, E3 -82315.720}
SPL {X  -157.725, Y  +355.675, Z    +0.000, E1  +284.959, E3 -82412.678}
SPL {X  -142.593, Y  +309.947, Z    +0.000, E1  +282.426, E3 -82406.342}
SPL {X  -142.198, Y  +309.176, Z    +0.000, E1  +283.218, E3 -82415.150}
ENDSPLINE

SPLINE
SPL {X  -142.352, Y  +309.474, Z    +0.000, E1  +284.206, E3 -82424.844}
ENDSPLINE

SPLINE
SPL {X  -141.929, Y  +308.657, Z    +0.000, E1  +285.131, E3 -82433.929}
SPL {X  -140.635, Y  +306.221, Z    +0.000, E1  +286.163, E3 -82444.342}
SPL {X  -138.743, Y  +302.832, Z    +0.000, E1  +287.062, E3 -82453.351}
SPL {X  -135.531, Y  +297.482, Z    +0.000, E1  +287.444, E3 -82459.186}
SPL {X  -132.271, Y  +292.493, Z    +0.000, E1  +287.844, E3 -82464.704}
SPL {X  -128.837, Y  +287.643, Z    +0.000, E1  +288.283, E3 -82470.142}
SPL {X  -124.965, Y  +282.598, Z    +0.000, E1  +288.800, E3 -82475.804}
SPL {X  -120.791, Y  +277.589, Z    +0.000, E1  +289.397, E3 -82481.376}
SPL {X   -74.058, Y  +240.683, Z    +0.000, E1  +305.011, E3 -82638.439}
ENDSPLINE

SPLINE
SPL {X  -130.401, Y  +289.805, Z    +0.000, E1  +307.505, E3 -82795.410}
SPL {X  -152.244, Y  +333.323, Z    +0.000, E1  +320.871, E3 -82812.222}
SPL {X  -158.218, Y  +358.753, Z    +0.000, E1  +336.397, E3 -82816.394}
SPL {X  -159.681, Y  +372.564, Z    +0.000, E1  +347.981, E3 -82817.446}
SPL {X  -159.987, Y  +381.561, Z    +0.000, E1  +356.806, E3 -82817.742}
SPL {X  -159.990, Y  +384.668, Z    +0.000, E1  +360.183, E3 -82817.768}
SPL {X  -159.990, Y  +389.080, Z    +0.000, E1  +370.094, E3 -82817.848}
SPL {X  -159.990, Y  +394.652, Z    +0.000, E1  +384.399, E3 -82818.097}
SPL {X  -159.990, Y  +401.914, Z    +0.000, E1  +400.147, E3 -82818.712}
SPL {X  -159.990, Y  +414.609, Z    +0.000, E1  +416.791, E3 -82820.449}
SPL {X  -159.990, Y  +464.476, Z    +0.000, E1  +431.765, E3 -82833.250}
SPL {X  -158.553, Y  +692.895, Z    +0.000, E1  +434.809, E3 -82932.013}
SPL {X  -156.740, Y  +703.585, Z    +0.000, E1  +434.640, E3 -82940.018}
SPL {X  -154.470, Y  +713.164, Z    +0.000, E1  +434.425, E3 -82947.853}
SPL {X  -152.098, Y  +721.129, Z    +0.000, E1  +434.190, E3 -82954.825}
SPL {X  -148.128, Y  +731.956, Z    +0.000, E1  +433.814, E3 -82964.906}
SPL {X  -143.804, Y  +741.622, Z    +0.000, E1  +433.324, E3 -82974.682}
SPL {X  -140.603, Y  +747.839, Z    +0.000, E1  +432.964, E3 -82981.198}
SPL {X  -137.184, Y  +753.824, Z    +0.000, E1  +432.574, E3 -82987.635}
SPL {X  -133.762, Y  +759.276, Z    +0.000, E1  +432.150, E3 -82993.688}
SPL {X  -130.927, Y  +763.451, Z    +0.000, E1  +431.785, E3 -82998.383}
SPL {X  -128.105, Y  +767.343, Z    +0.000, E1  +431.419, E3 -83002.772}
SPL {X  -124.554, Y  +771.914, Z    +0.000, E1  +430.935, E3 -83007.943}
SPL {X  -120.892, Y  +776.295, Z    +0.000, E1  +430.404, E3 -83012.827}
SPL {X  -118.039, Y  +779.498, Z    +0.000, E1  +429.949, E3 -83016.345}
SPL {X   -71.966, Y  +814.391, Z    +0.000, E1  +415.783, E3 -83154.997}
ENDSPLINE

